Yaskawa INFORM job: DEMO_ROOF_SIDE_0625_3PAINT_33.JBI

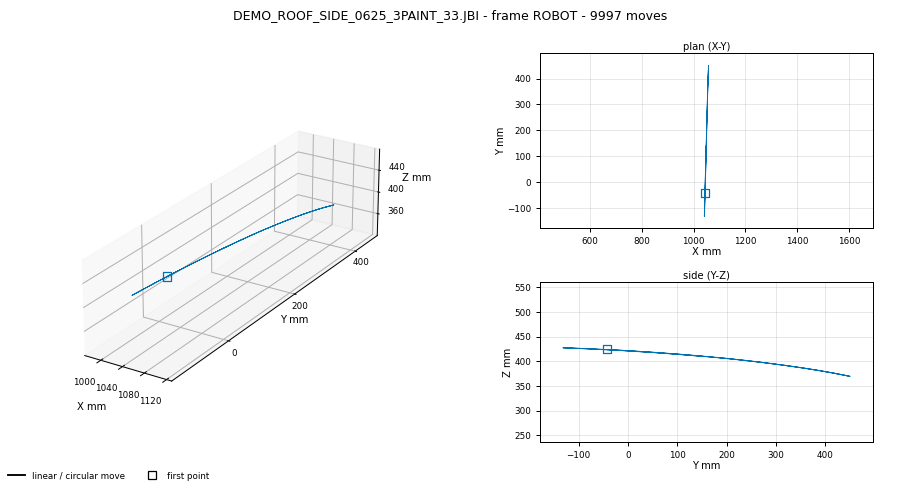
[picture p0: tool path of DEMO_ROOF_SIDE_0625_3PAINT_33.JBI in frame ROBOT, 9997 of 9997 moves have a stored position in this frame; points joined in program order, loops and branches not executed]
/JOB
//NAME DEMO_ROOF_SIDE_0625_3PAINT33
//POS
///NPOS 9997,0,0,0,0,0
///TOOL 0
///USER 0
///POSTYPE ROBOT
///RECTAN
///RCONF 1,0,0,0,0,0,0,0,0,0,0,0,0,0,0,0,0,0,0,0,0,0,0,0
C00000=1044.636,-42.308,424.466,169.630,34.372,156.485
C00001=1044.642,-42.058,424.454,169.632,34.373,156.485
C00002=1044.648,-41.809,424.441,169.634,34.375,156.485
C00003=1044.655,-41.560,424.428,169.636,34.375,156.486
C00004=1044.661,-41.310,424.415,169.638,34.376,156.486
C00005=1044.667,-41.061,424.402,169.640,34.377,156.486
C00006=1044.674,-40.810,424.389,169.642,34.378,156.486
C00007=1044.680,-40.561,424.376,169.645,34.379,156.486
C00008=1044.687,-40.311,424.364,169.647,34.380,156.486
C00009=1044.693,-40.062,424.351,169.649,34.381,156.486
C00010=1044.699,-39.813,424.337,169.651,34.382,156.486
C00011=1044.706,-39.562,424.324,169.653,34.383,156.486
C00012=1044.712,-39.313,424.311,169.656,34.384,156.487
C00013=1044.718,-39.063,424.299,169.658,34.385,156.487
C00014=1044.725,-38.814,424.286,169.660,34.385,156.487
C00015=1044.731,-38.565,424.273,169.662,34.387,156.487
C00016=1044.738,-38.314,424.260,169.664,34.388,156.487
C00017=1044.744,-38.065,424.246,169.666,34.389,156.487
C00018=1044.749,-37.816,424.233,169.668,34.390,156.487
C00019=1044.755,-37.566,424.219,169.670,34.391,156.488
C00020=1044.761,-37.316,424.207,169.672,34.392,156.488
C00021=1044.768,-37.067,424.193,169.674,34.393,156.488
C00022=1044.774,-36.817,424.180,169.677,34.394,156.488
C00023=1044.781,-36.568,424.167,169.679,34.395,156.488
C00024=1044.787,-36.318,424.154,169.681,34.396,156.488
C00025=1044.793,-36.069,424.141,169.683,34.398,156.488
C00026=1044.800,-35.819,424.127,169.685,34.398,156.489
C00027=1044.806,-35.538,424.113,169.687,34.400,156.489
C00028=1044.813,-35.257,424.097,169.689,34.401,156.489
C00029=1044.820,-34.977,424.083,169.692,34.402,156.489
C00030=1044.828,-34.695,424.068,169.694,34.403,156.489
C00031=1044.834,-34.446,424.055,169.696,34.405,156.489
C00032=1044.840,-34.197,424.042,169.698,34.405,156.489
C00033=1044.846,-33.947,424.028,169.700,34.407,156.490
C00034=1044.852,-33.697,424.014,169.702,34.407,156.490
C00035=1044.858,-33.448,424.002,169.704,34.409,156.490
C00036=1044.864,-33.198,423.988,169.706,34.410,156.490
C00037=1044.871,-32.949,423.975,169.708,34.411,156.490
C00038=1044.878,-32.699,423.961,169.710,34.412,156.490
C00039=1044.884,-32.450,423.948,169.712,34.413,156.491
C00040=1044.890,-32.200,423.935,169.714,34.414,156.491
C00041=1044.897,-31.951,423.921,169.716,34.415,156.491
C00042=1044.903,-31.701,423.908,169.718,34.416,156.491
C00043=1044.909,-31.452,423.895,169.720,34.417,156.491
C00044=1044.915,-31.201,423.881,169.722,34.418,156.491
C00045=1044.921,-30.952,423.868,169.724,34.419,156.491
C00046=1044.927,-30.703,423.855,169.726,34.420,156.491
C00047=1044.934,-30.453,423.841,169.728,34.422,156.492
C00048=1044.940,-30.203,423.828,169.730,34.422,156.492
C00049=1044.947,-29.954,423.814,169.732,34.424,156.492
C00050=1044.953,-29.704,423.801,169.734,34.424,156.492
C00051=1044.960,-29.455,423.788,169.736,34.426,156.492
C00052=1044.966,-29.206,423.774,169.739,34.427,156.492
C00053=1044.972,-28.955,423.760,169.741,34.428,156.493
C00054=1044.978,-28.706,423.747,169.743,34.429,156.493
C00055=1044.984,-28.457,423.733,169.745,34.430,156.493
C00056=1044.991,-28.207,423.720,169.748,34.431,156.493
C00057=1044.997,-27.958,423.707,169.750,34.432,156.493
C00058=1045.004,-27.708,423.693,169.752,34.434,156.493
C00059=1045.010,-27.458,423.680,169.754,34.434,156.493
C00060=1045.017,-27.209,423.666,169.756,34.436,156.494
C00061=1045.023,-26.959,423.652,169.758,34.436,156.494
C00062=1045.029,-26.710,423.639,169.760,34.438,156.494
C00063=1045.035,-26.461,423.625,169.762,34.439,156.494
C00064=1045.042,-26.211,423.611,169.763,34.440,156.494
C00065=1045.048,-25.961,423.597,169.765,34.441,156.494
C00066=1045.054,-25.712,423.584,169.767,34.443,156.495
C00067=1045.060,-25.462,423.570,169.769,34.444,156.495
C00068=1045.066,-25.213,423.557,169.771,34.445,156.495
C00069=1045.073,-24.963,423.543,169.773,34.446,156.495
C00070=1045.079,-24.714,423.528,169.775,34.447,156.495
C00071=1045.085,-24.464,423.515,169.777,34.448,156.495
C00072=1045.091,-24.214,423.501,169.779,34.450,156.496
C00073=1045.097,-23.965,423.488,169.781,34.451,156.496
C00074=1045.104,-23.715,423.474,169.783,34.452,156.496
C00075=1045.110,-23.465,423.460,169.785,34.453,156.496
C00076=1045.116,-23.217,423.446,169.787,34.454,156.496
C00077=1045.123,-22.967,423.433,169.789,34.456,156.496
C00078=1045.128,-22.717,423.419,169.791,34.457,156.497
C00079=1045.135,-22.467,423.405,169.793,34.458,156.497
C00080=1045.141,-22.218,423.390,169.795,34.459,156.497
C00081=1045.148,-21.968,423.377,169.797,34.461,156.497
C00082=1045.154,-21.719,423.364,169.799,34.461,156.497
C00083=1045.160,-21.469,423.350,169.801,34.463,156.497
C00084=1045.167,-21.220,423.335,169.804,34.464,156.498
C00085=1045.172,-20.970,423.321,169.806,34.465,156.498
C00086=1045.179,-20.720,423.308,169.808,34.466,156.498
C00087=1045.186,-20.472,423.294,169.810,34.468,156.498
C00088=1045.192,-20.222,423.280,169.812,34.469,156.498
C00089=1045.198,-19.972,423.266,169.814,34.470,156.498
C00090=1045.204,-19.723,423.251,169.816,34.471,156.499
C00091=1045.211,-19.441,423.236,169.818,34.472,156.499
C00092=1045.218,-19.159,423.220,169.820,34.474,156.499
C00093=1045.225,-18.878,423.205,169.822,34.475,156.499
C00094=1045.232,-18.596,423.189,169.824,34.477,156.499
C00095=1045.239,-18.347,423.175,169.826,34.478,156.500
C00096=1045.245,-18.097,423.161,169.828,34.479,156.500
C00097=1045.252,-17.848,423.147,169.830,34.480,156.500
C00098=1045.258,-17.598,423.133,169.832,34.481,156.500
C00099=1045.264,-17.348,423.119,169.834,34.482,156.500
C00100=1045.271,-17.099,423.105,169.836,34.484,156.500
C00101=1045.277,-16.849,423.091,169.838,34.485,156.501
C00102=1045.284,-16.600,423.077,169.840,34.486,156.501
C00103=1045.290,-16.350,423.063,169.842,34.487,156.501
C00104=1045.296,-16.101,423.049,169.844,34.488,156.501
C00105=1045.303,-15.851,423.035,169.846,34.490,156.501
C00106=1045.308,-15.602,423.021,169.848,34.491,156.502
C00107=1045.316,-15.352,423.007,169.850,34.492,156.502
C00108=1045.322,-15.102,422.993,169.852,34.493,156.502
C00109=1045.327,-14.853,422.978,169.854,34.495,156.502
C00110=1045.334,-14.603,422.964,169.855,34.496,156.502
C00111=1045.340,-14.354,422.950,169.858,34.497,156.502
C00112=1045.346,-14.104,422.936,169.860,34.499,156.503
C00113=1045.353,-13.855,422.922,169.862,34.500,156.503
C00114=1045.359,-13.605,422.907,169.864,34.501,156.503
C00115=1045.365,-13.356,422.893,169.866,34.502,156.503
C00116=1045.372,-13.107,422.878,169.868,34.503,156.503
C00117=1045.378,-12.856,422.864,169.870,34.505,156.504
C00118=1045.383,-12.607,422.850,169.872,34.506,156.504
C00119=1045.390,-12.357,422.836,169.874,34.508,156.504
C00120=1045.396,-12.109,422.821,169.876,34.509,156.504
C00121=1045.402,-11.859,422.806,169.877,34.510,156.504
C00122=1045.409,-11.610,422.793,169.879,34.512,156.505
C00123=1045.415,-11.360,422.778,169.881,34.512,156.505
C00124=1045.421,-11.110,422.764,169.883,34.514,156.505
C00125=1045.428,-10.861,422.750,169.885,34.515,156.505
C00126=1045.434,-10.611,422.735,169.887,34.516,156.505
C00127=1045.440,-10.361,422.721,169.889,34.518,156.505
C00128=1045.447,-10.112,422.707,169.891,34.519,156.506
C00129=1045.453,-9.863,422.692,169.893,34.521,156.506
C00130=1045.459,-9.613,422.678,169.895,34.522,156.506
C00131=1045.466,-9.364,422.664,169.896,34.523,156.506
C00132=1045.472,-9.114,422.649,169.898,34.525,156.507
C00133=1045.478,-8.865,422.634,169.900,34.525,156.507
C00134=1045.484,-8.615,422.620,169.903,34.527,156.507
C00135=1045.491,-8.366,422.606,169.905,34.528,156.507
C00136=1045.497,-8.117,422.591,169.907,34.529,156.507
C00137=1045.503,-7.866,422.577,169.909,34.531,156.507
C00138=1045.510,-7.617,422.562,169.911,34.532,156.508
C00139=1045.516,-7.368,422.548,169.913,34.534,156.508
C00140=1045.522,-7.118,422.533,169.914,34.535,156.508
C00141=1045.528,-6.868,422.519,169.916,34.536,156.508
C00142=1045.535,-6.620,422.505,169.918,34.537,156.508
C00143=1045.541,-6.370,422.490,169.920,34.538,156.509
C00144=1045.548,-6.120,422.475,169.922,34.540,156.509
C00145=1045.555,-5.871,422.460,169.924,34.541,156.509
C00146=1045.560,-5.621,422.447,169.926,34.542,156.509
C00147=1045.566,-5.372,422.432,169.928,34.544,156.509
C00148=1045.573,-5.122,422.417,169.929,34.545,156.510
C00149=1045.580,-4.873,422.402,169.931,34.546,156.510
C00150=1045.586,-4.624,422.388,169.933,34.548,156.510
C00151=1045.592,-4.373,422.373,169.935,34.549,156.510
C00152=1045.598,-4.124,422.359,169.937,34.551,156.510
C00153=1045.605,-3.875,422.345,169.939,34.551,156.510
C00154=1045.611,-3.625,422.330,169.941,34.553,156.511
C00155=1045.618,-3.342,422.313,169.943,34.555,156.511
C00156=1045.626,-3.059,422.296,169.946,34.556,156.511
C00157=1045.632,-2.775,422.279,169.948,34.557,156.511
C00158=1045.639,-2.492,422.262,169.950,34.559,156.512
C00159=1045.646,-2.243,422.247,169.952,34.561,156.512
C00160=1045.651,-1.994,422.233,169.954,34.562,156.512
C00161=1045.658,-1.744,422.218,169.956,34.563,156.512
C00162=1045.664,-1.495,422.203,169.957,34.565,156.513
C00163=1045.671,-1.245,422.188,169.959,34.566,156.513
C00164=1045.676,-0.996,422.173,169.961,34.567,156.513
C00165=1045.683,-0.746,422.158,169.963,34.569,156.513
C00166=1045.689,-0.497,422.143,169.965,34.570,156.513
C00167=1045.696,-0.247,422.128,169.967,34.572,156.514
C00168=1045.701,0.002,422.114,169.968,34.573,156.514
C00169=1045.708,0.252,422.099,169.970,34.575,156.514
C00170=1045.713,0.502,422.083,169.972,34.576,156.514
C00171=1045.720,0.751,422.068,169.974,34.578,156.515
C00172=1045.726,1.000,422.054,169.976,34.579,156.515
C00173=1045.732,1.250,422.039,169.978,34.580,156.515
C00174=1045.738,1.500,422.024,169.979,34.582,156.515
C00175=1045.745,1.749,422.009,169.982,34.583,156.515
C00176=1045.750,1.998,421.994,169.984,34.584,156.516
C00177=1045.757,2.248,421.979,169.986,34.586,156.516
C00178=1045.763,2.497,421.965,169.988,34.588,156.516
C00179=1045.770,2.746,421.949,169.989,34.589,156.516
C00180=1045.776,2.996,421.934,169.991,34.590,156.517
C00181=1045.783,3.246,421.919,169.993,34.592,156.517
C00182=1045.788,3.495,421.904,169.995,34.593,156.517
C00183=1045.795,3.744,421.889,169.997,34.594,156.517
C00184=1045.801,3.994,421.874,169.999,34.596,156.517
C00185=1045.807,4.244,421.859,170.000,34.597,156.518
C00186=1045.814,4.493,421.843,170.002,34.598,156.518
C00187=1045.820,4.743,421.828,170.004,34.600,156.518
C00188=1045.826,4.992,421.814,170.006,34.601,156.518
C00189=1045.832,5.241,421.799,170.008,34.603,156.518
C00190=1045.839,5.491,421.784,170.009,34.604,156.519
C00191=1045.845,5.740,421.768,170.011,34.606,156.519
C00192=1045.852,5.990,421.753,170.013,34.607,156.519
C00193=1045.858,6.239,421.738,170.016,34.608,156.519
C00194=1045.864,6.489,421.723,170.018,34.610,156.520
C00195=1045.869,6.738,421.708,170.020,34.611,156.520
C00196=1045.876,6.987,421.693,170.021,34.612,156.520
C00197=1045.882,7.237,421.678,170.023,34.614,156.520
C00198=1045.889,7.487,421.663,170.025,34.615,156.520
C00199=1045.895,7.736,421.648,170.027,34.617,156.521
C00200=1045.902,7.985,421.632,170.029,34.618,156.521
C00201=1045.908,8.235,421.617,170.030,34.620,156.521
C00202=1045.915,8.485,421.602,170.032,34.621,156.521
C00203=1045.921,8.734,421.586,170.034,34.623,156.522
C00204=1045.927,8.984,421.571,170.036,34.624,156.522
C00205=1045.933,9.233,421.556,170.038,34.625,156.522
C00206=1045.940,9.482,421.540,170.039,34.627,156.522
C00207=1045.946,9.731,421.526,170.041,34.628,156.522
C00208=1045.952,9.981,421.511,170.043,34.629,156.523
C00209=1045.959,10.230,421.495,170.045,34.631,156.523
C00210=1045.965,10.480,421.480,170.047,34.633,156.523
C00211=1045.971,10.730,421.465,170.049,34.634,156.523
C00212=1045.978,10.979,421.449,170.051,34.635,156.524
C00213=1045.984,11.228,421.434,170.053,34.637,156.524
C00214=1045.990,11.478,421.419,170.055,34.638,156.524
C00215=1045.997,11.727,421.403,170.057,34.639,156.524
C00216=1046.004,11.977,421.388,170.058,34.641,156.524
C00217=1046.010,12.226,421.373,170.060,34.642,156.525
C00218=1046.016,12.476,421.357,170.062,34.643,156.525
C00219=1046.023,12.761,421.340,170.064,34.645,156.525
C00220=1046.031,13.046,421.322,170.066,34.647,156.525
C00221=1046.038,13.331,421.305,170.068,34.648,156.526
C00222=1046.045,13.616,421.287,170.070,34.650,156.526
C00223=1046.052,13.865,421.272,170.072,34.651,156.526
C00224=1046.058,14.115,421.257,170.074,34.653,156.526
C00225=1046.065,14.364,421.241,170.076,34.654,156.526
C00226=1046.070,14.614,421.226,170.077,34.655,156.527
C00227=1046.077,14.863,421.210,170.080,34.657,156.527
C00228=1046.083,15.113,421.194,170.082,34.659,156.527
C00229=1046.090,15.362,421.179,170.084,34.660,156.527
C00230=1046.096,15.611,421.163,170.085,34.661,156.528
C00231=1046.102,15.861,421.148,170.087,34.663,156.528
C00232=1046.109,16.110,421.132,170.089,34.665,156.528
C00233=1046.114,16.360,421.117,170.091,34.666,156.528
C00234=1046.121,16.609,421.101,170.092,34.667,156.529
C00235=1046.127,16.859,421.086,170.094,34.669,156.529
C00236=1046.133,17.108,421.070,170.096,34.671,156.529
C00237=1046.140,17.357,421.054,170.098,34.672,156.529
C00238=1046.146,17.607,421.038,170.099,34.673,156.530
C00239=1046.152,17.856,421.023,170.101,34.675,156.530
C00240=1046.159,18.107,421.008,170.103,34.677,156.530
C00241=1046.165,18.356,420.991,170.105,34.678,156.530
C00242=1046.172,18.605,420.976,170.106,34.679,156.530
C00243=1046.177,18.855,420.960,170.109,34.681,156.531
C00244=1046.184,19.104,420.944,170.111,34.682,156.531
C00245=1046.191,19.353,420.929,170.113,34.684,156.531
C00246=1046.197,19.603,420.913,170.114,34.685,156.531
C00247=1046.203,19.852,420.898,170.116,34.687,156.532
C00248=1046.209,20.101,420.881,170.118,34.688,156.532
C00249=1046.216,20.351,420.866,170.120,34.690,156.532
C00250=1046.221,20.600,420.850,170.121,34.691,156.532
C00251=1046.228,20.849,420.834,170.123,34.693,156.533
C00252=1046.234,21.099,420.818,170.125,34.695,156.533
C00253=1046.240,21.349,420.803,170.127,34.696,156.533
C00254=1046.246,21.598,420.787,170.128,34.697,156.533
C00255=1046.253,21.848,420.770,170.130,34.699,156.534
C00256=1046.260,22.097,420.755,170.132,34.700,156.534
C00257=1046.265,22.347,420.739,170.134,34.702,156.534
C00258=1046.272,22.596,420.723,170.135,34.703,156.534
C00259=1046.278,22.845,420.707,170.138,34.705,156.535
C00260=1046.285,23.094,420.692,170.140,34.706,156.535
C00261=1046.291,23.344,420.675,170.142,34.708,156.535
C00262=1046.296,23.594,420.660,170.143,34.709,156.535
C00263=1046.303,23.843,420.644,170.145,34.711,156.536
C00264=1046.310,24.093,420.627,170.147,34.712,156.536
C00265=1046.316,24.342,420.612,170.148,34.714,156.536
C00266=1046.322,24.591,420.596,170.150,34.716,156.536
C00267=1046.329,24.841,420.581,170.152,34.717,156.537
C00268=1046.334,25.090,420.564,170.154,34.718,156.537
C00269=1046.340,25.339,420.548,170.155,34.720,156.537
C00270=1046.347,25.588,420.532,170.157,34.722,156.537
C00271=1046.354,25.839,420.516,170.159,34.723,156.538
C00272=1046.360,26.088,420.500,170.161,34.724,156.538
C00273=1046.366,26.337,420.484,170.163,34.726,156.538
C00274=1046.373,26.586,420.468,170.165,34.728,156.538
C00275=1046.379,26.835,420.452,170.167,34.729,156.538
C00276=1046.385,27.085,420.436,170.168,34.730,156.539
C00277=1046.392,27.335,420.420,170.170,34.732,156.539
C00278=1046.398,27.584,420.404,170.172,34.734,156.539
C00279=1046.404,27.834,420.388,170.174,34.735,156.539
C00280=1046.410,28.083,420.372,170.175,34.737,156.540
C00281=1046.416,28.332,420.356,170.177,34.738,156.540
C00282=1046.423,28.582,420.339,170.179,34.740,156.540
C00283=1046.430,28.868,420.321,170.181,34.741,156.541
C00284=1046.438,29.155,420.302,170.183,34.743,156.541
C00285=1046.445,29.440,420.284,170.185,34.745,156.541
C00286=1046.451,29.727,420.265,170.187,34.747,156.541
C00287=1046.458,29.977,420.249,170.189,34.749,156.542
C00288=1046.464,30.226,420.233,170.191,34.750,156.542
C00289=1046.470,30.476,420.217,170.193,34.751,156.542
C00290=1046.476,30.725,420.200,170.194,34.753,156.542
C00291=1046.482,30.974,420.183,170.196,34.755,156.543
C00292=1046.490,31.224,420.167,170.198,34.756,156.543
C00293=1046.496,31.473,420.151,170.200,34.758,156.543
C00294=1046.502,31.722,420.135,170.201,34.759,156.543
C00295=1046.507,31.972,420.119,170.203,34.761,156.544
C00296=1046.514,32.222,420.102,170.205,34.763,156.544
C00297=1046.521,32.471,420.086,170.206,34.764,156.544
C00298=1046.527,32.720,420.070,170.208,34.766,156.545
C00299=1046.533,32.969,420.054,170.210,34.767,156.545
C00300=1046.539,33.219,420.037,170.212,34.768,156.545
C00301=1046.545,33.468,420.020,170.214,34.770,156.545
C00302=1046.552,33.717,420.005,170.216,34.772,156.545
C00303=1046.558,33.967,419.988,170.218,34.774,156.546
C00304=1046.565,34.217,419.972,170.219,34.775,156.546
C00305=1046.571,34.466,419.956,170.221,34.776,156.546
C00306=1046.577,34.715,419.939,170.223,34.778,156.547
C00307=1046.583,34.964,419.922,170.224,34.780,156.547
C00308=1046.590,35.214,419.906,170.226,34.781,156.547
C00309=1046.596,35.463,419.890,170.228,34.783,156.547
C00310=1046.602,35.713,419.874,170.229,34.784,156.548
C00311=1046.609,35.963,419.857,170.231,34.786,156.548
C00312=1046.615,36.211,419.840,170.233,34.788,156.548
C00313=1046.621,36.461,419.824,170.236,34.789,156.548
C00314=1046.628,36.710,419.808,170.237,34.791,156.549
C00315=1046.634,36.960,419.792,170.239,34.792,156.549
C00316=1046.640,37.208,419.775,170.241,34.793,156.549
C00317=1046.646,37.458,419.758,170.242,34.795,156.549
C00318=1046.653,37.708,419.742,170.244,34.797,156.550
C00319=1046.659,37.957,419.725,170.246,34.799,156.550
C00320=1046.665,38.206,419.709,170.247,34.800,156.550
C00321=1046.671,38.456,419.692,170.249,34.801,156.550
C00322=1046.677,38.705,419.676,170.251,34.803,156.551
C00323=1046.684,38.954,419.659,170.252,34.805,156.551
C00324=1046.690,39.204,419.642,170.254,34.807,156.551
C00325=1046.697,39.453,419.625,170.256,34.808,156.551
C00326=1046.702,39.702,419.609,170.258,34.810,156.552
C00327=1046.709,39.952,419.592,170.260,34.811,156.552
C00328=1046.715,40.201,419.575,170.262,34.813,156.552
C00329=1046.720,40.451,419.558,170.263,34.814,156.553
C00330=1046.727,40.701,419.542,170.265,34.816,156.553
C00331=1046.733,40.949,419.525,170.267,34.818,156.553
C00332=1046.739,41.199,419.509,170.268,34.820,156.553
C00333=1046.746,41.448,419.491,170.270,34.821,156.554
C00334=1046.752,41.698,419.475,170.272,34.822,156.554
C00335=1046.758,41.947,419.459,170.273,34.824,156.554
C00336=1046.765,42.196,419.441,170.275,34.825,156.554
C00337=1046.771,42.446,419.425,170.277,34.827,156.555
C00338=1046.777,42.694,419.408,170.279,34.829,156.555
C00339=1046.784,42.944,419.391,170.281,34.831,156.555
C00340=1046.790,43.193,419.375,170.283,34.832,156.555
C00341=1046.796,43.443,419.358,170.285,34.834,156.556
C00342=1046.802,43.692,419.340,170.286,34.835,156.556
C00343=1046.808,43.942,419.324,170.288,34.837,156.556
C00344=1046.815,44.191,419.307,170.289,34.839,156.557
C00345=1046.820,44.441,419.290,170.291,34.840,156.557
C00346=1046.826,44.689,419.273,170.293,34.842,156.557
C00347=1046.833,44.977,419.253,170.295,34.844,156.558
C00348=1046.840,45.263,419.233,170.297,34.846,156.558
C00349=1046.848,45.549,419.215,170.298,34.848,156.558
C00350=1046.855,45.835,419.195,170.301,34.850,156.558
C00351=1046.861,46.085,419.178,170.303,34.852,156.559
C00352=1046.867,46.334,419.161,170.305,34.854,156.559
C00353=1046.873,46.583,419.144,170.306,34.855,156.559
C00354=1046.879,46.833,419.126,170.308,34.857,156.560
C00355=1046.885,47.082,419.109,170.310,34.858,156.560
C00356=1046.891,47.331,419.093,170.311,34.860,156.560
C00357=1046.897,47.581,419.075,170.313,34.861,156.560
C00358=1046.904,47.830,419.058,170.314,34.863,156.561
C00359=1046.910,48.080,419.042,170.316,34.865,156.561
C00360=1046.916,48.329,419.024,170.318,34.867,156.561
C00361=1046.922,48.578,419.007,170.320,34.868,156.562
C00362=1046.928,48.827,418.990,170.322,34.870,156.562
C00363=1046.934,49.076,418.973,170.324,34.872,156.562
C00364=1046.941,49.326,418.956,170.325,34.873,156.562
C00365=1046.947,49.575,418.939,170.327,34.875,156.563
C00366=1046.953,49.825,418.921,170.329,34.876,156.563
C00367=1046.959,50.074,418.904,170.330,34.878,156.563
C00368=1046.966,50.324,418.888,170.332,34.880,156.564
C00369=1046.971,50.573,418.870,170.334,34.882,156.564
C00370=1046.978,50.822,418.853,170.335,34.883,156.564
C00371=1046.984,51.071,418.836,170.337,34.885,156.564
C00372=1046.990,51.321,418.819,170.340,34.887,156.565
C00373=1046.996,51.570,418.802,170.341,34.888,156.565
C00374=1047.003,51.819,418.784,170.343,34.890,156.565
C00375=1047.009,52.068,418.767,170.344,34.891,156.565
C00376=1047.015,52.318,418.751,170.346,34.893,156.566
C00377=1047.021,52.568,418.733,170.348,34.895,156.566
C00378=1047.028,52.817,418.715,170.349,34.896,156.566
C00379=1047.034,53.066,418.698,170.351,34.898,156.567
C00380=1047.040,53.315,418.680,170.353,34.900,156.567
C00381=1047.046,53.565,418.664,170.354,34.902,156.567
C00382=1047.053,53.814,418.647,170.356,34.903,156.567
C00383=1047.058,54.063,418.629,170.359,34.905,156.568
C00384=1047.065,54.313,418.612,170.360,34.906,156.568
C00385=1047.071,54.562,418.594,170.362,34.908,156.568
C00386=1047.078,54.811,418.577,170.364,34.909,156.568
C00387=1047.084,55.060,418.560,170.365,34.911,156.569
C00388=1047.090,55.310,418.543,170.367,34.913,156.569
C00389=1047.096,55.559,418.526,170.369,34.915,156.569
C00390=1047.103,55.808,418.508,170.370,34.916,156.570
C00391=1047.109,56.058,418.491,170.372,34.918,156.570
C00392=1047.115,56.307,418.474,170.374,34.919,156.570
C00393=1047.121,56.557,418.456,170.375,34.921,156.570
C00394=1047.128,56.805,418.439,170.377,34.922,156.571
C00395=1047.134,57.055,418.421,170.379,34.924,156.571
C00396=1047.140,57.304,418.404,170.381,34.926,156.571
C00397=1047.147,57.553,418.386,170.383,34.928,156.572
C00398=1047.153,57.804,418.369,170.384,34.929,156.572
C00399=1047.159,58.052,418.352,170.386,34.931,156.572
C00400=1047.166,58.302,418.335,170.388,34.932,156.572
C00401=1047.171,58.551,418.317,170.389,34.934,156.573
C00402=1047.178,58.800,418.300,170.391,34.935,156.573
C00403=1047.184,59.050,418.282,170.393,34.937,156.573
C00404=1047.190,59.299,418.265,170.394,34.939,156.573
C00405=1047.197,59.548,418.247,170.397,34.941,156.574
C00406=1047.203,59.798,418.230,170.399,34.942,156.574
C00407=1047.210,60.047,418.213,170.400,34.944,156.574
C00408=1047.216,60.296,418.195,170.402,34.945,156.575
C00409=1047.223,60.546,418.178,170.404,34.947,156.575
C00410=1047.228,60.795,418.160,170.405,34.948,156.575
C00411=1047.236,61.081,418.140,170.407,34.950,156.575
C00412=1047.244,61.366,418.120,170.409,34.952,156.576
C00413=1047.251,61.652,418.100,170.411,34.954,156.576
C00414=1047.258,61.939,418.079,170.413,34.956,156.576
C00415=1047.264,62.188,418.062,170.415,34.958,156.577
C00416=1047.271,62.438,418.044,170.417,34.959,156.577
C00417=1047.278,62.687,418.027,170.419,34.961,156.577
C00418=1047.283,62.936,418.010,170.420,34.963,156.578
C00419=1047.290,63.185,417.992,170.422,34.964,156.578
C00420=1047.296,63.435,417.974,170.424,34.966,156.578
C00421=1047.303,63.684,417.956,170.425,34.967,156.578
C00422=1047.309,63.933,417.939,170.427,34.969,156.579
C00423=1047.316,64.182,417.921,170.429,34.970,156.579
C00424=1047.322,64.432,417.903,170.430,34.972,156.579
C00425=1047.327,64.681,417.886,170.432,34.974,156.579
C00426=1047.334,64.931,417.868,170.434,34.976,156.580
C00427=1047.341,65.180,417.850,170.436,34.978,156.580
C00428=1047.346,65.429,417.832,170.438,34.979,156.580
C00429=1047.352,65.679,417.814,170.440,34.981,156.581
C00430=1047.359,65.928,417.797,170.441,34.982,156.581
C00431=1047.365,66.177,417.779,170.443,34.984,156.581
C00432=1047.371,66.426,417.761,170.444,34.986,156.581
C00433=1047.378,66.676,417.743,170.446,34.987,156.582
C00434=1047.384,66.925,417.725,170.448,34.989,156.582
C00435=1047.389,67.174,417.708,170.449,34.990,156.582
C00436=1047.396,67.423,417.689,170.451,34.992,156.583
C00437=1047.403,67.673,417.672,170.454,34.994,156.583
C00438=1047.408,67.922,417.654,170.455,34.996,156.583
C00439=1047.415,68.171,417.636,170.457,34.998,156.583
C00440=1047.421,68.421,417.618,170.458,34.999,156.584
C00441=1047.428,68.670,417.600,170.460,35.001,156.584
C00442=1047.433,68.919,417.582,170.462,35.003,156.584
C00443=1047.440,69.168,417.564,170.463,35.004,156.585
C00444=1047.446,69.418,417.546,170.465,35.006,156.585
C00445=1047.453,69.667,417.528,170.467,35.008,156.585
C00446=1047.458,69.916,417.511,170.468,35.009,156.585
C00447=1047.465,70.166,417.493,170.471,35.011,156.586
C00448=1047.471,70.415,417.474,170.473,35.013,156.586
C00449=1047.476,70.664,417.457,170.474,35.014,156.586
C00450=1047.483,70.913,417.438,170.476,35.016,156.587
C00451=1047.489,71.163,417.420,170.477,35.018,156.587
C00452=1047.495,71.413,417.402,170.479,35.019,156.587
C00453=1047.502,71.661,417.384,170.481,35.021,156.588
C00454=1047.508,71.910,417.366,170.482,35.023,156.588
C00455=1047.514,72.159,417.348,170.484,35.025,156.588
C00456=1047.520,72.409,417.330,170.486,35.027,156.588
C00457=1047.526,72.658,417.312,170.488,35.028,156.589
C00458=1047.532,72.907,417.294,170.490,35.030,156.589
C00459=1047.539,73.157,417.275,170.491,35.032,156.589
C00460=1047.545,73.406,417.257,170.493,35.034,156.590
C00461=1047.551,73.655,417.238,170.495,35.035,156.590
C00462=1047.557,73.904,417.221,170.496,35.037,156.590
C00463=1047.563,74.154,417.202,170.498,35.039,156.591
C00464=1047.569,74.403,417.184,170.500,35.040,156.591
C00465=1047.576,74.652,417.166,170.501,35.042,156.591
C00466=1047.583,74.902,417.148,170.504,35.044,156.591
C00467=1047.588,75.150,417.130,170.505,35.045,156.592
C00468=1047.595,75.400,417.112,170.507,35.047,156.592
C00469=1047.601,75.649,417.093,170.509,35.049,156.592
C00470=1047.607,75.899,417.075,170.510,35.050,156.593
C00471=1047.614,76.148,417.057,170.512,35.052,156.593
C00472=1047.620,76.398,417.039,170.514,35.054,156.593
C00473=1047.626,76.646,417.021,170.515,35.056,156.594
C00474=1047.632,76.895,417.002,170.517,35.057,156.594
C00475=1047.639,77.182,416.982,170.519,35.059,156.594
C00476=1047.646,77.468,416.960,170.522,35.061,156.595
C00477=1047.653,77.753,416.939,170.523,35.063,156.595
C00478=1047.660,78.039,416.918,170.525,35.065,156.595
C00479=1047.667,78.288,416.899,170.527,35.067,156.596
C00480=1047.673,78.538,416.881,170.529,35.068,156.596
C00481=1047.679,78.786,416.863,170.530,35.070,156.596
C00482=1047.684,79.036,416.844,170.532,35.072,156.596
C00483=1047.691,79.286,416.826,170.533,35.074,156.597
C00484=1047.697,79.535,416.807,170.535,35.075,156.597
C00485=1047.703,79.784,416.789,170.538,35.077,156.597
C00486=1047.710,80.033,416.770,170.539,35.079,156.598
C00487=1047.715,80.282,416.752,170.541,35.081,156.598
C00488=1047.721,80.531,416.733,170.543,35.083,156.598
C00489=1047.728,80.781,416.715,170.544,35.084,156.599
C00490=1047.734,81.030,416.696,170.546,35.086,156.599
C00491=1047.740,81.279,416.678,170.547,35.088,156.599
C00492=1047.746,81.529,416.659,170.549,35.090,156.599
C00493=1047.752,81.778,416.640,170.551,35.092,156.600
C00494=1047.759,82.027,416.621,170.553,35.093,156.600
C00495=1047.764,82.276,416.604,170.555,35.095,156.600
C00496=1047.771,82.525,416.585,170.556,35.097,156.601
C00497=1047.777,82.774,416.567,170.558,35.099,156.601
C00498=1047.783,83.024,416.547,170.560,35.100,156.601
C00499=1047.789,83.273,416.529,170.561,35.102,156.602
C00500=1047.796,83.522,416.510,170.563,35.104,156.602
C00501=1047.802,83.772,416.492,170.565,35.106,156.602
C00502=1047.807,84.021,416.473,170.566,35.107,156.603
C00503=1047.814,84.270,416.454,170.569,35.109,156.603
C00504=1047.820,84.519,416.436,170.571,35.111,156.603
C00505=1047.826,84.768,416.417,170.572,35.113,156.603
C00506=1047.832,85.017,416.399,170.574,35.115,156.604
C00507=1047.838,85.266,416.379,170.575,35.116,156.604
C00508=1047.845,85.516,416.361,170.577,35.118,156.604
C00509=1047.851,85.765,416.343,170.579,35.120,156.605
C00510=1047.857,86.014,416.324,170.580,35.122,156.605
C00511=1047.863,86.264,416.305,170.582,35.123,156.605
C00512=1047.869,86.513,416.286,170.585,35.125,156.606
C00513=1047.876,86.762,416.268,170.586,35.127,156.606
C00514=1047.882,87.011,416.249,170.588,35.128,156.606
C00515=1047.888,87.261,416.230,170.589,35.130,156.607
C00516=1047.894,87.510,416.211,170.591,35.132,156.607
C00517=1047.901,87.759,416.192,170.593,35.133,156.607
C00518=1047.907,88.008,416.174,170.594,35.135,156.607
C00519=1047.913,88.257,416.155,170.596,35.137,156.608
C00520=1047.919,88.507,416.136,170.598,35.139,156.608
C00521=1047.926,88.756,416.117,170.600,35.140,156.608
C00522=1047.932,89.005,416.099,170.602,35.142,156.609
C00523=1047.938,89.254,416.079,170.604,35.144,156.609
C00524=1047.944,89.503,416.061,170.605,35.145,156.609
C00525=1047.951,89.753,416.042,170.607,35.147,156.610
C00526=1047.957,90.002,416.023,170.609,35.149,156.610
C00527=1047.963,90.251,416.004,170.610,35.150,156.610
C00528=1047.969,90.500,415.986,170.612,35.152,156.610
C00529=1047.975,90.750,415.966,170.613,35.154,156.611
C00530=1047.981,90.999,415.948,170.616,35.156,156.611
C00531=1047.987,91.248,415.928,170.618,35.158,156.611
C00532=1047.993,91.497,415.910,170.619,35.159,156.612
C00533=1047.999,91.747,415.891,170.621,35.161,156.612
C00534=1048.006,91.995,415.871,170.623,35.163,156.612
C00535=1048.011,92.245,415.852,170.624,35.165,156.613
C00536=1048.018,92.494,415.833,170.626,35.167,156.613
C00537=1048.024,92.743,415.814,170.627,35.168,156.613
C00538=1048.030,92.992,415.795,170.630,35.170,156.614
C00539=1048.037,93.278,415.773,170.632,35.172,156.614
C00540=1048.045,93.564,415.751,170.634,35.175,156.614
C00541=1048.051,93.849,415.729,170.636,35.177,156.615
C00542=1048.058,94.136,415.707,170.638,35.179,156.615
C00543=1048.064,94.385,415.689,170.639,35.180,156.615
C00544=1048.070,94.634,415.669,170.641,35.182,156.616
C00545=1048.077,94.883,415.650,170.643,35.184,156.616
C00546=1048.082,95.133,415.631,170.645,35.186,156.616
C00547=1048.089,95.382,415.612,170.647,35.187,156.617
C00548=1048.095,95.630,415.592,170.648,35.189,156.617
C00549=1048.101,95.880,415.573,170.650,35.191,156.617
C00550=1048.107,96.129,415.554,170.652,35.193,156.618
C00551=1048.114,96.379,415.535,170.653,35.194,156.618
C00552=1048.120,96.628,415.515,170.655,35.196,156.618
C00553=1048.126,96.877,415.497,170.657,35.198,156.619
C00554=1048.132,97.126,415.477,170.658,35.200,156.619
C00555=1048.138,97.376,415.458,170.661,35.201,156.619
C00556=1048.144,97.624,415.439,170.663,35.203,156.619
C00557=1048.150,97.874,415.419,170.664,35.205,156.620
C00558=1048.156,98.123,415.401,170.666,35.207,156.620
C00559=1048.162,98.371,415.381,170.668,35.209,156.620
C00560=1048.170,98.621,415.362,170.669,35.210,156.621
C00561=1048.175,98.871,415.343,170.671,35.212,156.621
C00562=1048.182,99.119,415.323,170.673,35.214,156.621
C00563=1048.188,99.369,415.304,170.675,35.216,156.622
C00564=1048.194,99.617,415.284,170.677,35.217,156.622
C00565=1048.200,99.867,415.265,170.678,35.219,156.622
C00566=1048.206,100.116,415.246,170.680,35.221,156.623
C00567=1048.213,100.365,415.226,170.682,35.223,156.623
C00568=1048.219,100.615,415.207,170.683,35.224,156.623
C00569=1048.224,100.864,415.188,170.685,35.226,156.624
C00570=1048.230,101.113,415.168,170.687,35.228,156.624
C00571=1048.237,101.362,415.149,170.689,35.230,156.624
C00572=1048.243,101.611,415.129,170.691,35.232,156.625
C00573=1048.249,101.860,415.110,170.693,35.234,156.625
C00574=1048.255,102.110,415.090,170.694,35.235,156.625
C00575=1048.261,102.359,415.071,170.696,35.237,156.625
C00576=1048.268,102.608,415.051,170.698,35.239,156.626
C00577=1048.273,102.857,415.032,170.699,35.241,156.626
C00578=1048.279,103.106,415.012,170.701,35.243,156.626
C00579=1048.285,103.355,414.993,170.704,35.245,156.627
C00580=1048.291,103.604,414.973,170.705,35.247,156.627
C00581=1048.298,103.854,414.954,170.707,35.249,156.628
C00582=1048.304,104.103,414.934,170.708,35.250,156.628
C00583=1048.310,104.352,414.914,170.710,35.252,156.628
C00584=1048.316,104.601,414.895,170.712,35.254,156.628
C00585=1048.322,104.850,414.875,170.713,35.256,156.629
C00586=1048.327,105.099,414.855,170.715,35.257,156.629
C00587=1048.335,105.349,414.836,170.718,35.259,156.629
C00588=1048.340,105.598,414.816,170.719,35.261,156.630
C00589=1048.346,105.847,414.796,170.721,35.263,156.630
C00590=1048.352,106.096,414.777,170.723,35.265,156.630
C00591=1048.358,106.345,414.757,170.724,35.266,156.631
C00592=1048.365,106.595,414.737,170.726,35.268,156.631
C00593=1048.371,106.843,414.718,170.728,35.270,156.631
C00594=1048.377,107.093,414.698,170.729,35.272,156.632
C00595=1048.383,107.341,414.678,170.732,35.273,156.632
C00596=1048.390,107.591,414.658,170.734,35.275,156.632
C00597=1048.395,107.840,414.639,170.735,35.277,156.633
C00598=1048.401,108.089,414.619,170.737,35.279,156.633
C00599=1048.407,108.338,414.599,170.739,35.281,156.633
C00600=1048.414,108.588,414.580,170.740,35.283,156.634
C00601=1048.420,108.837,414.560,170.742,35.284,156.634
C00602=1048.426,109.085,414.540,170.744,35.286,156.634
C00603=1048.433,109.371,414.517,170.747,35.289,156.635
C00604=1048.440,109.657,414.495,170.749,35.291,156.635
C00605=1048.447,109.943,414.472,170.751,35.292,156.635
C00606=1048.455,110.229,414.449,170.752,35.294,156.636
C00607=1048.461,110.478,414.429,170.754,35.296,156.636
C00608=1048.467,110.728,414.410,170.756,35.298,156.636
C00609=1048.473,110.977,414.390,170.758,35.300,156.637
C00610=1048.479,111.225,414.370,170.760,35.302,156.637
C00611=1048.485,111.475,414.350,170.762,35.304,156.637
C00612=1048.491,111.724,414.330,170.764,35.305,156.638
C00613=1048.497,111.973,414.310,170.765,35.307,156.638
C00614=1048.503,112.222,414.290,170.767,35.309,156.638
C00615=1048.510,112.471,414.270,170.769,35.311,156.639
C00616=1048.516,112.720,414.250,170.770,35.313,156.639
C00617=1048.522,112.969,414.230,170.772,35.315,156.639
C00618=1048.528,113.219,414.210,170.775,35.317,156.640
C00619=1048.534,113.467,414.190,170.776,35.318,156.640
C00620=1048.540,113.717,414.171,170.778,35.320,156.640
C00621=1048.547,113.966,414.150,170.780,35.322,156.641
C00622=1048.553,114.215,414.130,170.781,35.324,156.641
C00623=1048.558,114.464,414.110,170.783,35.326,156.641
C00624=1048.564,114.713,414.090,170.785,35.328,156.642
C00625=1048.570,114.963,414.070,170.787,35.330,156.642
C00626=1048.576,115.212,414.049,170.789,35.332,156.642
C00627=1048.582,115.461,414.029,170.791,35.334,156.643
C00628=1048.588,115.710,414.009,170.792,35.336,156.643
C00629=1048.594,115.959,413.989,170.794,35.337,156.643
C00630=1048.599,116.208,413.968,170.796,35.339,156.644
C00631=1048.605,116.457,413.948,170.797,35.341,156.644
C00632=1048.612,116.706,413.928,170.800,35.343,156.645
C00633=1048.618,116.955,413.908,170.802,35.345,156.645
C00634=1048.623,117.204,413.887,170.803,35.347,156.645
C00635=1048.630,117.454,413.867,170.805,35.349,156.646
C00636=1048.636,117.703,413.847,170.807,35.351,156.646
C00637=1048.641,117.952,413.827,170.808,35.353,156.646
C00638=1048.648,118.201,413.806,170.810,35.354,156.647
C00639=1048.654,118.450,413.786,170.813,35.356,156.647
C00640=1048.660,118.698,413.766,170.814,35.358,156.647
C00641=1048.666,118.948,413.745,170.816,35.360,156.648
C00642=1048.672,119.197,413.725,170.818,35.362,156.648
C00643=1048.679,119.446,413.704,170.820,35.363,156.648
C00644=1048.684,119.696,413.684,170.821,35.365,156.649
C00645=1048.690,119.944,413.664,170.823,35.367,156.649
C00646=1048.696,120.194,413.644,170.825,35.369,156.649
C00647=1048.702,120.443,413.624,170.827,35.371,156.650
C00648=1048.708,120.692,413.603,170.829,35.373,156.650
C00649=1048.715,120.941,413.582,170.831,35.375,156.650
C00650=1048.721,121.189,413.562,170.832,35.377,156.651
C00651=1048.726,121.439,413.541,170.834,35.378,156.651
C00652=1048.732,121.688,413.521,170.836,35.380,156.651
C00653=1048.738,121.937,413.501,170.838,35.382,156.652
C00654=1048.745,122.186,413.480,170.840,35.384,156.652
C00655=1048.751,122.435,413.460,170.842,35.386,156.652
C00656=1048.757,122.684,413.439,170.844,35.388,156.653
C00657=1048.762,122.934,413.419,170.845,35.390,156.653
C00658=1048.769,123.183,413.398,170.847,35.392,156.653
C00659=1048.775,123.431,413.378,170.849,35.394,156.654
C00660=1048.781,123.681,413.357,170.851,35.396,156.654
C00661=1048.787,123.930,413.337,170.853,35.397,156.654
C00662=1048.793,124.179,413.317,170.855,35.399,156.655
C00663=1048.799,124.428,413.295,170.857,35.401,156.655
C00664=1048.805,124.677,413.275,170.858,35.403,156.655
C00665=1048.812,124.926,413.255,170.860,35.405,156.656
C00666=1048.817,125.175,413.234,170.862,35.407,156.656
C00667=1048.825,125.462,413.210,170.864,35.409,156.656
C00668=1048.832,125.747,413.187,170.867,35.411,156.657
C00669=1048.839,126.032,413.163,170.869,35.413,156.657
C00670=1048.846,126.318,413.139,170.871,35.415,156.658
C00671=1048.852,126.567,413.119,170.873,35.417,156.658
C00672=1048.858,126.816,413.099,170.874,35.419,156.658
C00673=1048.864,127.065,413.078,170.876,35.421,156.659
C00674=1048.870,127.314,413.058,170.879,35.423,156.659
C00675=1048.876,127.564,413.037,170.881,35.425,156.659
C00676=1048.883,127.812,413.016,170.882,35.426,156.660
C00677=1048.889,128.062,412.996,170.884,35.428,156.660
C00678=1048.895,128.310,412.974,170.886,35.430,156.660
C00679=1048.901,128.560,412.954,170.888,35.432,156.661
C00680=1048.908,128.809,412.934,170.889,35.434,156.661
C00681=1048.914,129.058,412.912,170.892,35.436,156.661
C00682=1048.920,129.307,412.892,170.894,35.437,156.662
C00683=1048.926,129.555,412.871,170.896,35.439,156.662
C00684=1048.932,129.805,412.851,170.897,35.441,156.662
C00685=1048.938,130.054,412.831,170.899,35.443,156.663
C00686=1048.944,130.303,412.809,170.901,35.445,156.663
C00687=1048.951,130.553,412.789,170.903,35.447,156.663
C00688=1048.957,130.801,412.768,170.905,35.449,156.664
C00689=1048.963,131.051,412.747,170.907,35.450,156.664
C00690=1048.970,131.299,412.726,170.909,35.452,156.664
C00691=1048.975,131.549,412.705,170.911,35.454,156.665
C00692=1048.982,131.798,412.684,170.912,35.456,156.665
C00693=1048.988,132.047,412.664,170.914,35.458,156.665
C00694=1048.994,132.296,412.642,170.916,35.460,156.666
C00695=1049.000,132.544,412.622,170.919,35.462,156.666
C00696=1049.006,132.794,412.601,170.920,35.464,156.666
C00697=1049.011,133.042,412.579,170.922,35.466,156.667
C00698=1049.018,133.292,412.559,170.924,35.467,156.667
C00699=1049.024,133.541,412.537,170.926,35.469,156.667
C00700=1049.030,133.790,412.516,170.927,35.471,156.668
C00701=1049.036,134.039,412.496,170.929,35.474,156.668
C00702=1049.042,134.288,412.474,170.932,35.476,156.669
C00703=1049.048,134.537,412.453,170.934,35.477,156.669
C00704=1049.054,134.786,412.433,170.935,35.479,156.669
C00705=1049.060,135.035,412.411,170.937,35.481,156.670
C00706=1049.066,135.284,412.390,170.939,35.483,156.670
C00707=1049.072,135.533,412.370,170.941,35.485,156.670
C00708=1049.079,135.782,412.348,170.944,35.487,156.671
C00709=1049.085,136.031,412.326,170.945,35.489,156.671
C00710=1049.091,136.280,412.306,170.947,35.491,156.671
C00711=1049.097,136.529,412.285,170.949,35.493,156.672
C00712=1049.102,136.778,412.264,170.951,35.494,156.672
C00713=1049.109,137.027,412.242,170.952,35.496,156.672
C00714=1049.115,137.277,412.222,170.954,35.498,156.673
C00715=1049.121,137.525,412.200,170.957,35.500,156.673
C00716=1049.127,137.774,412.179,170.959,35.502,156.674
C00717=1049.133,138.024,412.157,170.961,35.504,156.674
C00718=1049.139,138.272,412.137,170.962,35.506,156.674
C00719=1049.145,138.522,412.115,170.964,35.508,156.675
C00720=1049.151,138.771,412.094,170.966,35.510,156.675
C00721=1049.157,139.019,412.073,170.969,35.512,156.675
C00722=1049.164,139.268,412.051,170.970,35.514,156.676
C00723=1049.170,139.518,412.031,170.972,35.516,156.676
C00724=1049.175,139.766,412.009,170.974,35.518,156.676
C00725=1049.181,140.016,411.988,170.976,35.520,156.677
C00726=1049.188,140.265,411.966,170.978,35.521,156.677
C00727=1049.193,140.513,411.945,170.979,35.524,156.678
C00728=1049.199,140.763,411.923,170.982,35.526,156.678
C00729=1049.205,141.012,411.901,170.984,35.528,156.678
C00730=1049.212,141.260,411.881,170.986,35.530,156.679
C00731=1049.219,141.546,411.856,170.988,35.532,156.679
C00732=1049.225,141.831,411.831,170.990,35.534,156.679
C00733=1049.232,142.117,411.808,170.993,35.536,156.680
C00734=1049.239,142.403,411.782,170.995,35.539,156.680
C00735=1049.246,142.652,411.761,170.997,35.541,156.681
C00736=1049.251,142.900,411.739,170.999,35.543,156.681
C00737=1049.257,143.150,411.718,171.000,35.545,156.681
C00738=1049.263,143.399,411.696,171.002,35.546,156.682
C00739=1049.269,143.647,411.675,171.004,35.548,156.682
C00740=1049.275,143.896,411.653,171.007,35.550,156.682
C00741=1049.281,144.146,411.632,171.009,35.553,156.683
C00742=1049.287,144.395,411.610,171.010,35.555,156.683
C00743=1049.293,144.643,411.589,171.012,35.557,156.684
C00744=1049.299,144.893,411.567,171.014,35.558,156.684
C00745=1049.305,145.142,411.545,171.016,35.560,156.684
C00746=1049.312,145.391,411.524,171.019,35.562,156.685
C00747=1049.318,145.639,411.503,171.021,35.564,156.685
C00748=1049.324,145.888,411.481,171.022,35.567,156.685
C00749=1049.330,146.138,411.460,171.024,35.568,156.686
C00750=1049.336,146.387,411.438,171.026,35.570,156.686
C00751=1049.343,146.635,411.416,171.028,35.572,156.687
C00752=1049.348,146.884,411.395,171.031,35.574,156.687
C00753=1049.355,147.133,411.373,171.033,35.576,156.687
C00754=1049.361,147.382,411.351,171.034,35.578,156.688
C00755=1049.367,147.632,411.330,171.036,35.580,156.688
C00756=1049.373,147.881,411.308,171.038,35.582,156.688
C00757=1049.378,148.130,411.286,171.040,35.584,156.689
C00758=1049.384,148.378,411.264,171.043,35.586,156.689
C00759=1049.390,148.627,411.242,171.045,35.588,156.689
C00760=1049.397,148.877,411.220,171.046,35.590,156.690
C00761=1049.403,149.126,411.199,171.048,35.592,156.690
C00762=1049.408,149.374,411.178,171.050,35.594,156.691
C00763=1049.415,149.623,411.155,171.052,35.596,156.691
C00764=1049.421,149.872,411.134,171.055,35.598,156.691
C00765=1049.426,150.122,411.111,171.057,35.600,156.692
C00766=1049.433,150.371,411.090,171.058,35.602,156.692
C00767=1049.438,150.619,411.068,171.060,35.604,156.692
C00768=1049.445,150.868,411.046,171.062,35.607,156.693
C00769=1049.451,151.117,411.024,171.064,35.608,156.693
C00770=1049.456,151.366,411.002,171.067,35.610,156.694
C00771=1049.463,151.615,410.980,171.069,35.612,156.694
C00772=1049.469,151.864,410.958,171.071,35.615,156.694
C00773=1049.475,152.113,410.936,171.072,35.617,156.695
C00774=1049.481,152.361,410.915,171.074,35.618,156.695
C00775=1049.486,152.611,410.892,171.076,35.620,156.696
C00776=1049.493,152.860,410.870,171.079,35.623,156.696
C00777=1049.499,153.109,410.848,171.081,35.625,156.696
C00778=1049.505,153.358,410.827,171.083,35.627,156.697
C00779=1049.511,153.607,410.804,171.085,35.628,156.697
C00780=1049.517,153.856,410.782,171.087,35.631,156.698
C00781=1049.523,154.105,410.760,171.089,35.633,156.698
C00782=1049.529,154.353,410.739,171.091,35.635,156.698
C00783=1049.534,154.603,410.716,171.093,35.636,156.699
C00784=1049.541,154.851,410.694,171.095,35.639,156.699
C00785=1049.547,155.100,410.672,171.097,35.641,156.699
C00786=1049.554,155.349,410.650,171.099,35.643,156.700
C00787=1049.559,155.599,410.628,171.102,35.645,156.700
C00788=1049.565,155.847,410.605,171.104,35.647,156.701
C00789=1049.571,156.097,410.583,171.105,35.649,156.701
C00790=1049.577,156.345,410.561,171.107,35.651,156.701
C00791=1049.583,156.594,410.539,171.109,35.653,156.702
C00792=1049.589,156.843,410.516,171.111,35.655,156.702
C00793=1049.595,157.092,410.495,171.114,35.657,156.702
C00794=1049.601,157.340,410.473,171.116,35.660,156.703
C00795=1049.608,157.626,410.447,171.118,35.661,156.703
C00796=1049.615,157.911,410.421,171.120,35.664,156.704
C00797=1049.622,158.197,410.396,171.122,35.666,156.704
C00798=1049.629,158.481,410.370,171.126,35.669,156.705
C00799=1049.635,158.730,410.348,171.127,35.671,156.705
C00800=1049.641,158.979,410.325,171.129,35.673,156.705
C00801=1049.647,159.229,410.304,171.131,35.675,156.706
C00802=1049.653,159.477,410.281,171.133,35.677,156.706
C00803=1049.659,159.726,410.259,171.136,35.679,156.707
C00804=1049.665,159.975,410.237,171.138,35.681,156.707
C00805=1049.672,160.224,410.215,171.140,35.683,156.707
C00806=1049.677,160.473,410.192,171.142,35.685,156.708
C00807=1049.683,160.722,410.170,171.144,35.688,156.708
C00808=1049.689,160.971,410.147,171.146,35.689,156.709
C00809=1049.695,161.220,410.124,171.149,35.692,156.709
C00810=1049.701,161.469,410.101,171.150,35.694,156.709
C00811=1049.706,161.718,410.079,171.152,35.696,156.710
C00812=1049.712,161.967,410.057,171.154,35.698,156.710
C00813=1049.718,162.216,410.034,171.156,35.701,156.711
C00814=1049.724,162.465,410.011,171.159,35.702,156.711
C00815=1049.729,162.714,409.988,171.161,35.705,156.711
C00816=1049.736,162.963,409.966,171.163,35.707,156.712
C00817=1049.742,163.212,409.943,171.165,35.709,156.712
C00818=1049.747,163.460,409.920,171.167,35.711,156.713
C00819=1049.753,163.709,409.897,171.170,35.714,156.713
C00820=1049.759,163.957,409.875,171.171,35.716,156.714
C00821=1049.765,164.206,409.852,171.173,35.718,156.714
C00822=1049.770,164.456,409.830,171.175,35.720,156.714
C00823=1049.776,164.705,409.807,171.177,35.722,156.715
C00824=1049.782,164.953,409.784,171.180,35.725,156.715
C00825=1049.788,165.202,409.762,171.182,35.727,156.716
C00826=1049.794,165.451,409.739,171.184,35.729,156.716
C00827=1049.799,165.700,409.716,171.186,35.731,156.716
C00828=1049.806,165.949,409.693,171.188,35.733,156.717
C00829=1049.812,166.198,409.670,171.191,35.735,156.717
C00830=1049.818,166.447,409.647,171.193,35.738,156.718
C00831=1049.824,166.696,409.624,171.195,35.740,156.718
C00832=1049.829,166.945,409.601,171.197,35.742,156.719
C00833=1049.835,167.194,409.578,171.199,35.744,156.719
C00834=1049.841,167.442,409.556,171.202,35.746,156.719
C00835=1049.847,167.691,409.533,171.203,35.748,156.720
C00836=1049.853,167.940,409.510,171.205,35.751,156.720
C00837=1049.859,168.189,409.487,171.207,35.753,156.721
C00838=1049.865,168.438,409.464,171.209,35.755,156.721
C00839=1049.870,168.687,409.441,171.212,35.757,156.721
C00840=1049.877,168.935,409.419,171.214,35.759,156.722
C00841=1049.882,169.184,409.396,171.216,35.762,156.722
C00842=1049.888,169.433,409.373,171.218,35.764,156.723
C00843=1049.895,169.683,409.350,171.220,35.766,156.723
C00844=1049.900,169.932,409.327,171.223,35.768,156.724
C00845=1049.906,170.180,409.304,171.225,35.771,156.724
C00846=1049.912,170.429,409.282,171.227,35.772,156.724
C00847=1049.918,170.678,409.259,171.229,35.775,156.725
C00848=1049.924,170.926,409.235,171.231,35.777,156.725
C00849=1049.930,171.175,409.212,171.234,35.779,156.726
C00850=1049.936,171.425,409.189,171.236,35.781,156.726
C00851=1049.942,171.674,409.166,171.238,35.784,156.726
C00852=1049.949,171.922,409.143,171.240,35.785,156.727
C00853=1049.954,172.171,409.121,171.242,35.788,156.727
C00854=1049.960,172.419,409.097,171.245,35.790,156.728
C00855=1049.966,172.668,409.074,171.247,35.792,156.728
C00856=1049.972,172.918,409.051,171.249,35.795,156.729
C00857=1049.978,173.167,409.028,171.251,35.797,156.729
C00858=1049.984,173.416,409.005,171.253,35.799,156.729
C00859=1049.991,173.699,408.978,171.256,35.802,156.730
C00860=1049.998,173.985,408.952,171.259,35.804,156.730
C00861=1050.005,174.269,408.925,171.261,35.807,156.731
C00862=1050.012,174.554,408.899,171.263,35.809,156.731
C00863=1050.017,174.803,408.876,171.265,35.811,156.732
C00864=1050.024,175.052,408.853,171.268,35.813,156.732
C00865=1050.031,175.301,408.829,171.270,35.816,156.733
C00866=1050.036,175.550,408.806,171.272,35.818,156.733
C00867=1050.042,175.798,408.783,171.274,35.820,156.733
C00868=1050.048,176.047,408.760,171.277,35.822,156.734
C00869=1050.054,176.296,408.736,171.280,35.824,156.734
C00870=1050.060,176.545,408.713,171.282,35.826,156.735
C00871=1050.066,176.794,408.690,171.284,35.829,156.735
C00872=1050.072,177.042,408.667,171.286,35.831,156.735
C00873=1050.079,177.292,408.644,171.289,35.833,156.736
C00874=1050.085,177.540,408.620,171.291,35.836,156.736
C00875=1050.091,177.789,408.598,171.293,35.837,156.737
C00876=1050.097,178.038,408.574,171.295,35.840,156.737
C00877=1050.103,178.287,408.551,171.297,35.842,156.738
C00878=1050.109,178.536,408.528,171.300,35.844,156.738
C00879=1050.115,178.785,408.504,171.302,35.846,156.738
C00880=1050.121,179.034,408.481,171.304,35.849,156.739
C00881=1050.127,179.282,408.457,171.306,35.850,156.739
C00882=1050.134,179.531,408.434,171.308,35.853,156.740
C00883=1050.140,179.779,408.411,171.311,35.855,156.740
C00884=1050.146,180.028,408.388,171.313,35.857,156.741
C00885=1050.153,180.277,408.364,171.316,35.860,156.741
C00886=1050.158,180.526,408.341,171.318,35.861,156.741
C00887=1050.165,180.775,408.317,171.320,35.864,156.742
C00888=1050.171,181.024,408.294,171.323,35.866,156.742
C00889=1050.177,181.272,408.270,171.325,35.868,156.743
C00890=1050.183,181.522,408.247,171.327,35.871,156.743
C00891=1050.189,181.770,408.223,171.329,35.873,156.744
C00892=1050.196,182.020,408.200,171.332,35.875,156.744
C00893=1050.202,182.268,408.176,171.334,35.877,156.744
C00894=1050.208,182.516,408.152,171.336,35.879,156.745
C00895=1050.214,182.766,408.129,171.339,35.882,156.745
C00896=1050.220,183.014,408.105,171.341,35.884,156.746
C00897=1050.226,183.264,408.082,171.344,35.886,156.746
C00898=1050.233,183.512,408.059,171.346,35.888,156.747
C00899=1050.240,183.761,408.035,171.348,35.890,156.747
C00900=1050.245,184.010,408.012,171.350,35.893,156.748
C00901=1050.251,184.258,407.988,171.352,35.895,156.748
C00902=1050.257,184.507,407.964,171.355,35.897,156.748
C00903=1050.262,184.756,407.940,171.357,35.900,156.749
C00904=1050.268,185.005,407.917,171.359,35.902,156.749
C00905=1050.274,185.254,407.892,171.361,35.905,156.750
C00906=1050.280,185.502,407.868,171.365,35.907,156.750
C00907=1050.286,185.751,407.844,171.367,35.909,156.751
C00908=1050.292,186.000,407.821,171.369,35.912,156.751
C00909=1050.298,186.249,407.797,171.371,35.914,156.752
C00910=1050.304,186.498,407.773,171.374,35.916,156.752
C00911=1050.310,186.746,407.749,171.376,35.919,156.753
C00912=1050.315,186.995,407.725,171.378,35.921,156.753
C00913=1050.322,187.244,407.701,171.380,35.924,156.753
C00914=1050.327,187.492,407.676,171.383,35.926,156.754
C00915=1050.333,187.741,407.653,171.385,35.929,156.754
C00916=1050.339,187.991,407.629,171.388,35.931,156.755
C00917=1050.345,188.239,407.605,171.390,35.933,156.755
C00918=1050.351,188.488,407.580,171.392,35.936,156.756
C00919=1050.357,188.736,407.557,171.395,35.938,156.756
C00920=1050.363,188.986,407.532,171.397,35.941,156.757
C00921=1050.369,189.234,407.509,171.399,35.943,156.757
C00922=1050.374,189.483,407.484,171.401,35.945,156.758
C00923=1050.381,189.767,407.457,171.405,35.948,156.758
C00924=1050.388,190.052,407.429,171.407,35.951,156.759
C00925=1050.395,190.336,407.402,171.410,35.954,156.759
C00926=1050.402,190.620,407.374,171.413,35.956,156.760
C00927=1050.408,190.869,407.350,171.415,35.959,156.760
C00928=1050.414,191.118,407.325,171.417,35.961,156.761
C00929=1050.419,191.366,407.301,171.420,35.963,156.761
C00930=1050.426,191.615,407.277,171.422,35.966,156.762
C00931=1050.431,191.864,407.253,171.425,35.968,156.762
C00932=1050.438,192.113,407.229,171.427,35.971,156.763
C00933=1050.443,192.361,407.205,171.429,35.973,156.763
C00934=1050.450,192.610,407.181,171.431,35.976,156.764
C00935=1050.455,192.859,407.156,171.435,35.978,156.764
C00936=1050.462,193.108,407.132,171.437,35.981,156.765
C00937=1050.467,193.356,407.108,171.439,35.983,156.765
C00938=1050.474,193.605,407.083,171.441,35.986,156.766
C00939=1050.479,193.853,407.059,171.444,35.988,156.766
C00940=1050.485,194.103,407.034,171.446,35.990,156.767
C00941=1050.492,194.352,407.010,171.449,35.993,156.767
C00942=1050.497,194.600,406.986,171.451,35.995,156.768
C00943=1050.504,194.849,406.962,171.454,35.998,156.768
C00944=1050.510,195.097,406.937,171.456,36.000,156.769
C00945=1050.516,195.346,406.913,171.458,36.002,156.769
C00946=1050.522,195.595,406.889,171.461,36.005,156.769
C00947=1050.528,195.844,406.865,171.464,36.007,156.770
C00948=1050.534,196.092,406.840,171.466,36.009,156.770
C00949=1050.540,196.341,406.816,171.468,36.012,156.771
C00950=1050.546,196.590,406.791,171.470,36.014,156.771
C00951=1050.552,196.839,406.767,171.474,36.017,156.772
C00952=1050.558,197.087,406.742,171.476,36.019,156.772
C00953=1050.564,197.336,406.718,171.478,36.022,156.773
C00954=1050.571,197.585,406.694,171.480,36.024,156.773
C00955=1050.577,197.833,406.669,171.484,36.027,156.774
C00956=1050.583,198.082,406.645,171.486,36.029,156.774
C00957=1050.589,198.331,406.620,171.488,36.031,156.775
C00958=1050.595,198.579,406.595,171.490,36.034,156.775
C00959=1050.601,198.828,406.571,171.494,36.036,156.776
C00960=1050.607,199.078,406.546,171.496,36.039,156.776
C00961=1050.614,199.325,406.522,171.498,36.042,156.777
C00962=1050.620,199.575,406.497,171.500,36.044,156.777
C00963=1050.625,199.824,406.473,171.504,36.047,156.778
C00964=1050.632,200.072,406.448,171.506,36.049,156.778
C00965=1050.638,200.321,406.424,171.508,36.052,156.779
C00966=1050.645,200.569,406.399,171.510,36.054,156.779
C00967=1050.651,200.818,406.374,171.514,36.056,156.780
C00968=1050.657,201.067,406.349,171.516,36.059,156.780
C00969=1050.663,201.315,406.325,171.518,36.061,156.781
C00970=1050.669,201.564,406.300,171.520,36.064,156.781
C00971=1050.675,201.813,406.275,171.524,36.066,156.782
C00972=1050.681,202.062,406.250,171.526,36.069,156.782
C00973=1050.687,202.310,406.226,171.528,36.072,156.783
C00974=1050.693,202.559,406.201,171.531,36.074,156.783
C00975=1050.699,202.808,406.176,171.534,36.077,156.784
C00976=1050.705,203.056,406.151,171.536,36.079,156.784
C00977=1050.711,203.305,406.126,171.538,36.081,156.785
C00978=1050.717,203.554,406.102,171.541,36.084,156.785
C00979=1050.723,203.803,406.076,171.544,36.087,156.786
C00980=1050.729,204.051,406.051,171.546,36.089,156.786
C00981=1050.735,204.300,406.027,171.548,36.092,156.787
C00982=1050.741,204.549,406.001,171.552,36.095,156.787
C00983=1050.747,204.797,405.976,171.554,36.097,156.788
C00984=1050.752,205.046,405.952,171.556,36.100,156.788
C00985=1050.759,205.294,405.927,171.559,36.103,156.789
C00986=1050.766,205.543,405.902,171.562,36.105,156.789
C00987=1050.790,206.596,405.796,171.789,36.201,156.808
C00988=1050.797,206.846,405.769,171.790,36.205,156.809
C00989=1050.804,207.098,405.743,171.793,36.208,156.809
C00990=1050.810,207.349,405.717,171.795,36.211,156.810
C00991=1050.817,207.600,405.691,171.797,36.215,156.811
C00992=1050.824,207.849,405.664,171.799,36.218,156.812
C00993=1050.829,208.098,405.638,171.801,36.221,156.812
C00994=1050.836,208.346,405.612,171.803,36.225,156.813
C00995=1050.843,208.594,405.586,171.805,36.228,156.814
C00996=1050.849,208.843,405.559,171.806,36.232,156.814
C00997=1050.855,209.092,405.534,171.809,36.235,156.815
C00998=1050.862,209.340,405.507,171.811,36.238,156.816
C00999=1050.869,209.588,405.481,171.813,36.242,156.816
C01000=1050.874,209.837,405.455,171.815,36.245,156.817
C01001=1050.881,210.086,405.429,171.816,36.248,156.818
C01002=1050.888,210.334,405.403,171.819,36.252,156.819
C01003=1050.893,210.582,405.376,171.821,36.256,156.819
C01004=1050.901,210.831,405.350,171.823,36.259,156.820
C01005=1050.906,211.080,405.324,171.825,36.262,156.821
C01006=1050.913,211.329,405.298,171.827,36.266,156.821
C01007=1050.920,211.577,405.272,171.829,36.269,156.822
C01008=1050.925,211.825,405.245,171.831,36.272,156.823
C01009=1050.933,212.074,405.218,171.832,36.275,156.823
C01010=1050.938,212.322,405.192,171.835,36.279,156.824
C01011=1050.945,212.570,405.166,171.837,36.283,156.825
C01012=1050.951,212.820,405.139,171.839,36.286,156.825
C01013=1050.957,213.068,405.113,171.841,36.289,156.826
C01014=1050.964,213.317,405.086,171.843,36.293,156.827
C01015=1050.970,213.565,405.060,171.845,36.296,156.828
C01016=1050.976,213.814,405.034,171.847,36.299,156.828
C01017=1050.983,214.062,405.007,171.850,36.303,156.829
C01018=1050.989,214.311,404.981,171.851,36.306,156.830
C01019=1050.996,214.560,404.954,171.853,36.310,156.830
C01020=1051.002,214.808,404.928,171.856,36.313,156.831
C01021=1051.008,215.056,404.901,171.857,36.316,156.832
C01022=1051.015,215.305,404.874,171.860,36.320,156.832
C01023=1051.021,215.553,404.848,171.862,36.323,156.833
C01024=1051.028,215.802,404.821,171.863,36.326,156.834
C01025=1051.033,216.050,404.795,171.866,36.330,156.835
C01026=1051.041,216.299,404.768,171.868,36.333,156.835
C01027=1051.046,216.548,404.742,171.870,36.337,156.836
C01028=1051.053,216.796,404.714,171.872,36.340,156.837
C01029=1051.059,217.044,404.688,171.874,36.343,156.837
C01030=1051.066,217.293,404.661,171.877,36.347,156.838
C01031=1051.072,217.541,404.635,171.878,36.350,156.839
C01032=1051.079,217.790,404.608,171.881,36.353,156.839
C01033=1051.085,218.038,404.582,171.883,36.357,156.840
C01034=1051.092,218.287,404.555,171.884,36.360,156.841
C01035=1051.097,218.536,404.528,171.887,36.364,156.842
C01036=1051.105,218.784,404.501,171.889,36.366,156.842
C01037=1051.111,219.032,404.474,171.891,36.370,156.843
C01038=1051.118,219.281,404.448,171.893,36.373,156.844
C01039=1051.123,219.529,404.421,171.895,36.377,156.844
C01040=1051.130,219.778,404.394,171.898,36.380,156.845
C01041=1051.136,220.026,404.368,171.899,36.383,156.846
C01042=1051.143,220.275,404.340,171.902,36.387,156.846
C01043=1051.150,220.523,404.314,171.904,36.390,156.847
C01044=1051.156,220.780,404.286,171.906,36.393,156.848
C01045=1051.163,221.037,404.258,171.908,36.397,156.848
C01046=1051.169,221.294,404.231,171.910,36.400,156.849
C01047=1051.176,221.550,404.203,171.913,36.404,156.850
C01048=1051.182,221.798,404.176,171.915,36.407,156.851
C01049=1051.189,222.047,404.149,171.917,36.410,156.851
C01050=1051.194,222.296,404.122,171.919,36.414,156.852
C01051=1051.201,222.544,404.094,171.921,36.417,156.853
C01052=1051.207,222.792,404.068,171.924,36.420,156.853
C01053=1051.213,223.041,404.041,171.926,36.424,156.854
C01054=1051.221,223.290,404.014,171.927,36.427,156.855
C01055=1051.226,223.538,403.987,171.930,36.430,156.855
C01056=1051.233,223.786,403.959,171.932,36.434,156.856
C01057=1051.239,224.035,403.933,171.935,36.437,156.857
C01058=1051.245,224.283,403.905,171.936,36.441,156.858
C01059=1051.252,224.532,403.878,171.938,36.444,156.858
C01060=1051.258,224.780,403.852,171.941,36.447,156.859
C01061=1051.265,225.029,403.824,171.943,36.451,156.860
C01062=1051.271,225.277,403.797,171.945,36.454,156.860
C01063=1051.278,225.526,403.770,171.947,36.457,156.861
C01064=1051.284,225.775,403.743,171.949,36.460,156.862
C01065=1051.290,226.022,403.715,171.952,36.464,156.862
C01066=1051.296,226.271,403.688,171.954,36.467,156.863
C01067=1051.303,226.520,403.661,171.956,36.470,156.864
C01068=1051.310,226.768,403.634,171.958,36.473,156.864
C01069=1051.316,227.016,403.607,171.961,36.477,156.865
C01070=1051.323,227.265,403.579,171.963,36.480,156.866
C01071=1051.329,227.513,403.552,171.965,36.484,156.867
C01072=1051.335,227.762,403.525,171.968,36.487,156.867
C01073=1051.342,228.011,403.498,171.969,36.490,156.868
C01074=1051.348,228.258,403.470,171.972,36.493,156.869
C01075=1051.354,228.507,403.443,171.974,36.497,156.869
C01076=1051.361,228.756,403.416,171.976,36.500,156.870
C01077=1051.368,229.004,403.388,171.979,36.503,156.871
C01078=1051.373,229.253,403.361,171.980,36.506,156.871
C01079=1051.380,229.501,403.333,171.983,36.510,156.872
C01080=1051.387,229.750,403.306,171.985,36.513,156.873
C01081=1051.393,229.997,403.278,171.987,36.516,156.873
C01082=1051.399,230.246,403.251,171.990,36.520,156.874
C01083=1051.406,230.495,403.224,171.992,36.523,156.875
C01084=1051.412,230.743,403.196,171.994,36.526,156.875
C01085=1051.419,230.991,403.168,171.996,36.529,156.876
C01086=1051.425,231.240,403.141,171.999,36.533,156.877
C01087=1051.430,231.488,403.114,172.001,36.536,156.877
C01088=1051.437,231.737,403.086,172.003,36.540,156.878
C01089=1051.444,231.985,403.058,172.006,36.543,156.879
C01090=1051.450,232.233,403.030,172.008,36.546,156.880
C01091=1051.456,232.482,403.004,172.010,36.550,156.880
C01092=1051.463,232.730,402.976,172.012,36.553,156.881
C01093=1051.469,232.979,402.948,172.014,36.556,156.882
C01094=1051.475,233.227,402.920,172.017,36.559,156.882
C01095=1051.481,233.475,402.893,172.019,36.563,156.883
C01096=1051.488,233.724,402.865,172.022,36.566,156.884
C01097=1051.495,233.972,402.837,172.024,36.569,156.885
C01098=1051.501,234.221,402.809,172.027,36.573,156.885
C01099=1051.507,234.469,402.781,172.028,36.576,156.886
C01100=1051.514,234.718,402.754,172.030,36.579,156.887
C01101=1051.520,234.967,402.726,172.033,36.582,156.887
C01102=1051.526,235.216,402.699,172.035,36.586,156.888
C01103=1051.533,235.466,402.670,172.038,36.589,156.889
C01104=1051.539,235.714,402.642,172.040,36.592,156.889
C01105=1051.545,235.962,402.614,172.043,36.596,156.890
C01106=1051.551,236.211,402.587,172.045,36.599,156.891
C01107=1051.558,236.459,402.559,172.047,36.603,156.892
C01108=1051.565,236.707,402.531,172.049,36.606,156.892
C01109=1051.571,236.956,402.503,172.051,36.609,156.893
C01110=1051.577,237.205,402.475,172.054,36.612,156.894
C01111=1051.583,237.452,402.448,172.056,36.616,156.894
C01112=1051.589,237.701,402.419,172.058,36.619,156.895
C01113=1051.596,237.950,402.392,172.061,36.622,156.896
C01114=1051.603,238.198,402.364,172.063,36.625,156.896
C01115=1051.609,238.446,402.336,172.066,36.629,156.897
C01116=1051.616,238.695,402.307,172.068,36.632,156.898
C01117=1051.622,238.943,402.279,172.071,36.635,156.898
C01118=1051.628,239.191,402.252,172.073,36.638,156.899
C01119=1051.634,239.439,402.224,172.075,36.642,156.900
C01120=1051.641,239.688,402.196,172.078,36.645,156.900
C01121=1051.648,239.936,402.168,172.080,36.648,156.901
C01122=1051.654,240.185,402.139,172.083,36.651,156.902
C01123=1051.661,240.433,402.111,172.085,36.655,156.903
C01124=1051.667,240.682,402.083,172.088,36.658,156.903
C01125=1051.673,240.930,402.055,172.089,36.661,156.904
C01126=1051.680,241.178,402.027,172.091,36.664,156.905
C01127=1051.686,241.427,401.999,172.094,36.668,156.905
C01128=1051.693,241.675,401.971,172.096,36.671,156.906
C01129=1051.698,241.923,401.943,172.099,36.674,156.907
C01130=1051.705,242.171,401.915,172.101,36.677,156.907
C01131=1051.711,242.420,401.886,172.104,36.681,156.908
C01132=1051.718,242.668,401.858,172.106,36.684,156.909
C01133=1051.724,242.916,401.829,172.108,36.687,156.910
C01134=1051.730,243.165,401.801,172.111,36.691,156.910
C01135=1051.737,243.413,401.773,172.113,36.694,156.911
C01136=1051.743,243.662,401.744,172.116,36.697,156.912
C01137=1051.750,243.910,401.717,172.118,36.700,156.912
C01138=1051.756,244.158,401.688,172.121,36.704,156.913
C01139=1051.763,244.407,401.660,172.123,36.707,156.914
C01140=1051.769,244.655,401.631,172.126,36.710,156.914
C01141=1051.775,244.904,401.602,172.128,36.714,156.915
C01142=1051.782,245.151,401.574,172.130,36.717,156.916
C01143=1051.788,245.400,401.546,172.133,36.720,156.917
C01144=1051.794,245.648,401.517,172.135,36.723,156.917
C01145=1051.801,245.897,401.489,172.138,36.727,156.918
C01146=1051.807,246.145,401.460,172.140,36.730,156.919
C01147=1051.812,246.393,401.432,172.143,36.733,156.919
C01148=1051.819,246.641,401.403,172.145,36.737,156.920
C01149=1051.826,246.889,401.374,172.147,36.740,156.921
C01150=1051.831,247.138,401.346,172.150,36.743,156.922
C01151=1051.838,247.386,401.317,172.152,36.747,156.922
C01152=1051.844,247.634,401.289,172.155,36.750,156.923
C01153=1051.850,247.883,401.260,172.157,36.754,156.924
C01154=1051.856,248.131,401.231,172.160,36.757,156.924
C01155=1051.862,248.380,401.202,172.162,36.760,156.925
C01156=1051.868,248.625,401.174,172.165,36.764,156.926
C01157=1051.875,248.870,401.145,172.167,36.767,156.926
C01158=1051.881,249.116,401.117,172.170,36.770,156.927
C01159=1051.888,249.362,401.088,172.172,36.773,156.928
C01160=1051.894,249.608,401.060,172.174,36.777,156.929
C01161=1051.900,249.854,401.031,172.177,36.780,156.929
C01162=1051.906,250.100,401.003,172.179,36.783,156.930
C01163=1051.913,250.345,400.974,172.182,36.787,156.931
C01164=1051.919,250.594,400.945,172.184,36.790,156.931
C01165=1051.925,250.842,400.916,172.188,36.793,156.932
C01166=1051.931,251.090,400.888,172.190,36.796,156.933
C01167=1051.937,251.339,400.859,172.193,36.800,156.934
C01168=1051.943,251.587,400.830,172.195,36.803,156.934
C01169=1051.950,251.834,400.801,172.197,36.806,156.935
C01170=1051.957,252.083,400.772,172.200,36.810,156.936
C01171=1051.964,252.331,400.743,172.202,36.813,156.936
C01172=1051.970,252.580,400.714,172.205,36.816,156.937
C01173=1051.976,252.828,400.686,172.207,36.819,156.938
C01174=1051.982,253.076,400.657,172.210,36.823,156.938
C01175=1051.988,253.325,400.628,172.212,36.826,156.939
C01176=1051.994,253.573,400.599,172.215,36.829,156.940
C01177=1052.001,253.821,400.570,172.218,36.833,156.941
C01178=1052.007,254.069,400.540,172.221,36.835,156.941
C01179=1052.015,254.318,400.512,172.223,36.839,156.942
C01180=1052.021,254.566,400.483,172.225,36.842,156.943
C01181=1052.027,254.814,400.454,172.228,36.845,156.943
C01182=1052.033,255.062,400.425,172.230,36.849,156.944
C01183=1052.040,255.310,400.396,172.233,36.852,156.945
C01184=1052.046,255.558,400.366,172.235,36.855,156.946
C01185=1052.053,255.807,400.337,172.239,36.858,156.946
C01186=1052.059,256.055,400.308,172.241,36.862,156.947
C01187=1052.065,256.303,400.279,172.244,36.865,156.948
C01188=1052.071,256.551,400.250,172.246,36.868,156.948
C01189=1052.078,256.800,400.221,172.249,36.871,156.949
C01190=1052.085,257.048,400.191,172.251,36.875,156.950
C01191=1052.091,257.297,400.162,172.253,36.878,156.950
C01192=1052.098,257.544,400.133,172.257,36.881,156.951
C01193=1052.104,257.792,400.104,172.259,36.884,156.952
C01194=1052.111,258.041,400.075,172.262,36.888,156.953
C01195=1052.117,258.289,400.046,172.264,36.891,156.953
C01196=1052.124,258.537,400.017,172.267,36.894,156.954
C01197=1052.131,258.786,399.987,172.269,36.898,156.955
C01198=1052.137,259.034,399.958,172.273,36.901,156.955
C01199=1052.143,259.281,399.929,172.275,36.904,156.956
C01200=1052.150,259.530,399.900,172.278,36.907,156.957
C01201=1052.156,259.778,399.870,172.280,36.911,156.958
C01202=1052.163,260.026,399.841,172.283,36.914,156.958
C01203=1052.169,260.274,399.811,172.286,36.917,156.959
C01204=1052.176,260.523,399.782,172.288,36.920,156.960
C01205=1052.182,260.771,399.753,172.291,36.924,156.960
C01206=1052.189,261.019,399.724,172.293,36.927,156.961
C01207=1052.196,261.267,399.694,172.296,36.930,156.962
C01208=1052.202,261.515,399.665,172.299,36.933,156.962
C01209=1052.208,261.764,399.636,172.302,36.936,156.963
C01210=1052.215,262.012,399.605,172.304,36.939,156.964
C01211=1052.222,262.260,399.576,172.307,36.943,156.965
C01212=1052.228,262.505,399.547,172.310,36.946,156.965
C01213=1052.235,262.750,399.519,172.313,36.949,156.966
C01214=1052.242,262.995,399.490,172.315,36.952,156.967
C01215=1052.248,263.240,399.459,172.318,36.956,156.967
C01216=1052.253,263.484,399.430,172.320,36.959,156.968
C01217=1052.260,263.729,399.401,172.324,36.962,156.969
C01218=1052.266,263.975,399.372,172.326,36.965,156.970
C01219=1052.273,264.219,399.342,172.328,36.969,156.970
C01220=1052.279,264.467,399.313,172.331,36.972,156.971
C01221=1052.285,264.715,399.283,172.333,36.975,156.972
C01222=1052.292,264.964,399.253,172.337,36.979,156.972
C01223=1052.298,265.211,399.224,172.339,36.982,156.973
C01224=1052.304,265.460,399.194,172.342,36.985,156.974
C01225=1052.311,265.708,399.164,172.344,36.989,156.975
C01226=1052.318,265.956,399.134,172.348,36.992,156.975
C01227=1052.324,266.205,399.104,172.350,36.995,156.976
C01228=1052.330,266.452,399.074,172.353,36.999,156.977
C01229=1052.337,266.700,399.045,172.355,37.002,156.978
C01230=1052.343,266.949,399.015,172.359,37.005,156.978
C01231=1052.349,267.196,398.985,172.361,37.008,156.979
C01232=1052.357,267.445,398.955,172.364,37.012,156.980
C01233=1052.362,267.693,398.925,172.366,37.015,156.980
C01234=1052.369,267.941,398.895,172.370,37.018,156.981
C01235=1052.375,268.189,398.865,172.372,37.021,156.982
C01236=1052.381,268.437,398.836,172.375,37.025,156.983
C01237=1052.388,268.686,398.805,172.378,37.028,156.983
C01238=1052.394,268.933,398.775,172.381,37.032,156.984
C01239=1052.401,269.182,398.744,172.383,37.035,156.985
C01240=1052.407,269.429,398.715,172.386,37.038,156.986
C01241=1052.414,269.678,398.685,172.389,37.042,156.986
C01242=1052.420,269.926,398.655,172.392,37.045,156.987
C01243=1052.427,270.174,398.625,172.394,37.048,156.988
C01244=1052.433,270.422,398.594,172.398,37.052,156.989
C01245=1052.439,270.670,398.564,172.400,37.055,156.989
C01246=1052.446,270.918,398.534,172.403,37.058,156.990
C01247=1052.452,271.166,398.503,172.406,37.062,156.991
C01248=1052.459,271.415,398.474,172.409,37.065,156.991
C01249=1052.465,271.663,398.444,172.411,37.068,156.992
C01250=1052.472,271.911,398.414,172.415,37.071,156.993
C01251=1052.478,272.159,398.383,172.417,37.075,156.994
C01252=1052.485,272.407,398.353,172.420,37.078,156.994
C01253=1052.491,272.655,398.323,172.423,37.081,156.995
C01254=1052.497,272.903,398.292,172.426,37.085,156.996
C01255=1052.504,273.151,398.262,172.428,37.088,156.997
C01256=1052.510,273.399,398.232,172.432,37.091,156.997
C01257=1052.516,273.648,398.201,172.434,37.095,156.998
C01258=1052.523,273.894,398.171,172.437,37.098,156.999
C01259=1052.529,274.143,398.140,172.440,37.102,157.000
C01260=1052.535,274.391,398.109,172.443,37.105,157.000
C01261=1052.542,274.639,398.079,172.445,37.108,157.001
C01262=1052.549,274.888,398.049,172.449,37.112,157.002
C01263=1052.555,275.135,398.018,172.451,37.115,157.003
C01264=1052.562,275.384,397.988,172.454,37.119,157.003
C01265=1052.568,275.631,397.958,172.457,37.122,157.004
C01266=1052.574,275.879,397.926,172.460,37.125,157.005
C01267=1052.580,276.127,397.896,172.463,37.128,157.006
C01268=1052.587,276.374,397.866,172.466,37.132,157.006
C01269=1052.594,276.621,397.836,172.468,37.135,157.007
C01270=1052.600,276.869,397.805,172.472,37.138,157.008
C01271=1052.606,277.115,397.775,172.474,37.142,157.009
C01272=1052.613,277.362,397.744,172.477,37.145,157.009
C01273=1052.619,277.609,397.713,172.480,37.149,157.010
C01274=1052.626,277.856,397.683,172.483,37.152,157.011
C01275=1052.633,278.103,397.652,172.486,37.155,157.012
C01276=1052.639,278.350,397.622,172.489,37.159,157.012
C01277=1052.645,278.599,397.591,172.491,37.162,157.013
C01278=1052.652,278.847,397.560,172.495,37.165,157.014
C01279=1052.658,279.095,397.529,172.497,37.169,157.014
C01280=1052.665,279.343,397.499,172.501,37.172,157.015
C01281=1052.671,279.591,397.468,172.503,37.176,157.016
C01282=1052.677,279.839,397.437,172.507,37.179,157.017
C01283=1052.684,280.087,397.406,172.510,37.182,157.018
C01284=1052.690,280.335,397.375,172.512,37.186,157.018
C01285=1052.696,280.582,397.344,172.516,37.189,157.019
C01286=1052.703,280.831,397.313,172.518,37.192,157.020
C01287=1052.710,281.079,397.282,172.522,37.196,157.021
C01288=1052.715,281.327,397.252,172.524,37.199,157.021
C01289=1052.722,281.574,397.220,172.527,37.203,157.022
C01290=1052.729,281.823,397.190,172.530,37.206,157.023
C01291=1052.735,282.070,397.158,172.533,37.210,157.024
C01292=1052.741,282.319,397.128,172.536,37.213,157.025
C01293=1052.748,282.567,397.096,172.539,37.217,157.025
C01294=1052.754,282.814,397.065,172.542,37.220,157.026
C01295=1052.760,283.062,397.035,172.545,37.224,157.027
C01296=1052.767,283.310,397.003,172.548,37.226,157.027
C01297=1052.774,283.558,396.972,172.551,37.230,157.028
C01298=1052.780,283.806,396.941,172.554,37.233,157.029
C01299=1052.786,284.054,396.910,172.557,37.237,157.030
C01300=1052.793,284.302,396.878,172.561,37.240,157.031
C01301=1052.800,284.550,396.848,172.563,37.244,157.031
C01302=1052.806,284.799,396.816,172.567,37.247,157.032
C01303=1052.812,285.046,396.785,172.569,37.251,157.033
C01304=1052.818,285.294,396.753,172.573,37.254,157.034
C01305=1052.825,285.542,396.723,172.575,37.258,157.035
C01306=1052.832,285.790,396.691,172.579,37.261,157.035
C01307=1052.838,286.038,396.660,172.581,37.265,157.036
C01308=1052.845,286.286,396.628,172.585,37.267,157.037
C01309=1052.851,286.533,396.597,172.587,37.271,157.038
C01310=1052.857,286.782,396.566,172.591,37.274,157.038
C01311=1052.864,287.029,396.535,172.594,37.278,157.039
C01312=1052.871,287.277,396.504,172.597,37.281,157.040
C01313=1052.878,287.525,396.472,172.600,37.285,157.041
C01314=1052.884,287.773,396.441,172.603,37.288,157.041
C01315=1052.891,288.021,396.409,172.606,37.292,157.042
C01316=1052.897,288.269,396.378,172.609,37.295,157.043
C01317=1052.903,288.516,396.346,172.612,37.299,157.044
C01318=1052.910,288.764,396.315,172.615,37.302,157.045
C01319=1052.917,289.012,396.283,172.618,37.306,157.045
C01320=1052.923,289.261,396.251,172.622,37.309,157.046
C01321=1052.929,289.508,396.220,172.624,37.312,157.047
C01322=1052.936,289.756,396.188,172.628,37.316,157.048
C01323=1052.943,290.004,396.157,172.631,37.319,157.049
C01324=1052.949,290.262,396.124,172.634,37.323,157.049
C01325=1052.956,290.519,396.091,172.637,37.327,157.050
C01326=1052.962,290.776,396.059,172.641,37.330,157.051
C01327=1052.970,291.032,396.026,172.644,37.334,157.052
C01328=1052.976,291.281,395.994,172.647,37.338,157.053
C01329=1052.982,291.529,395.962,172.650,37.341,157.053
C01330=1052.989,291.776,395.931,172.653,37.345,157.054
C01331=1052.995,292.025,395.899,172.657,37.348,157.055
C01332=1053.002,292.273,395.867,172.659,37.352,157.056
C01333=1053.009,292.520,395.835,172.663,37.355,157.057
C01334=1053.014,292.767,395.803,172.666,37.359,157.057
C01335=1053.021,293.015,395.772,172.669,37.362,157.058
C01336=1053.027,293.263,395.740,172.673,37.365,157.059
C01337=1053.034,293.511,395.708,172.675,37.369,157.060
C01338=1053.041,293.759,395.676,172.679,37.372,157.061
C01339=1053.047,294.007,395.644,172.681,37.376,157.061
C01340=1053.054,294.254,395.612,172.685,37.380,157.062
C01341=1053.060,294.502,395.581,172.689,37.383,157.063
C01342=1053.067,294.751,395.548,172.691,37.387,157.064
C01343=1053.074,294.998,395.516,172.695,37.390,157.065
C01344=1053.080,295.246,395.484,172.697,37.394,157.065
C01345=1053.087,295.494,395.453,172.701,37.397,157.066
C01346=1053.093,295.742,395.420,172.705,37.401,157.067
C01347=1053.100,295.990,395.389,172.707,37.404,157.068
C01348=1053.106,296.237,395.356,172.711,37.408,157.069
C01349=1053.113,296.485,395.324,172.714,37.411,157.070
C01350=1053.119,296.733,395.292,172.717,37.415,157.070
C01351=1053.125,296.981,395.260,172.720,37.419,157.071
C01352=1053.131,297.229,395.227,172.724,37.422,157.072
C01353=1053.138,297.476,395.195,172.727,37.426,157.073
C01354=1053.144,297.724,395.163,172.730,37.430,157.074
C01355=1053.151,297.972,395.130,172.733,37.433,157.075
C01356=1053.157,298.220,395.098,172.737,37.437,157.075
C01357=1053.163,298.468,395.065,172.740,37.441,157.076
C01358=1053.170,298.715,395.033,172.743,37.444,157.077
C01359=1053.176,298.963,395.001,172.746,37.448,157.078
C01360=1053.182,299.211,394.968,172.750,37.451,157.079
C01361=1053.188,299.458,394.936,172.753,37.455,157.080
C01362=1053.194,299.707,394.904,172.756,37.459,157.080
C01363=1053.202,299.954,394.871,172.760,37.462,157.081
C01364=1053.208,300.201,394.839,172.762,37.466,157.082
C01365=1053.215,300.450,394.806,172.766,37.470,157.083
C01366=1053.221,300.697,394.773,172.770,37.473,157.084
C01367=1053.227,300.946,394.741,172.772,37.477,157.085
C01368=1053.234,301.193,394.709,172.776,37.481,157.085
C01369=1053.240,301.440,394.676,172.779,37.484,157.086
C01370=1053.247,301.688,394.643,172.783,37.488,157.087
C01371=1053.253,301.936,394.610,172.786,37.492,157.088
C01372=1053.260,302.184,394.577,172.789,37.496,157.089
C01373=1053.266,302.432,394.545,172.793,37.499,157.090
C01374=1053.273,302.679,394.513,172.796,37.502,157.091
C01375=1053.279,302.927,394.480,172.799,37.506,157.091
C01376=1053.285,303.175,394.448,172.803,37.510,157.092
C01377=1053.292,303.422,394.415,172.806,37.514,157.093
C01378=1053.299,303.670,394.382,172.809,37.517,157.094
C01379=1053.305,303.918,394.349,172.813,37.521,157.095
C01380=1053.312,304.191,394.313,172.816,37.525,157.096
C01381=1053.320,304.464,394.277,172.820,37.529,157.097
C01382=1053.327,304.737,394.241,172.824,37.533,157.098
C01383=1053.334,305.010,394.205,172.827,37.537,157.099
C01384=1053.341,305.258,394.172,172.831,37.541,157.099
C01385=1053.347,305.505,394.139,172.835,37.545,157.100
C01386=1053.353,305.753,394.106,172.838,37.548,157.101
C01387=1053.361,306.001,394.074,172.841,37.552,157.102
C01388=1053.367,306.248,394.040,172.845,37.555,157.103
C01389=1053.374,306.496,394.008,172.848,37.559,157.104
C01390=1053.381,306.744,393.975,172.852,37.563,157.105
C01391=1053.387,306.991,393.942,172.856,37.567,157.106
C01392=1053.393,307.239,393.909,172.858,37.570,157.106
C01393=1053.400,307.487,393.876,172.862,37.574,157.107
C01394=1053.407,307.734,393.843,172.865,37.578,157.108
C01395=1053.414,307.982,393.810,172.869,37.582,157.109
C01396=1053.421,308.230,393.777,172.873,37.585,157.110
C01397=1053.427,308.478,393.745,172.875,37.589,157.111
C01398=1053.434,308.724,393.711,172.879,37.592,157.111
C01399=1053.440,308.973,393.678,172.883,37.596,157.112
C01400=1053.447,309.220,393.645,172.886,37.600,157.113
C01401=1053.454,309.469,393.612,172.890,37.604,157.114
C01402=1053.460,309.716,393.579,172.894,37.607,157.115
C01403=1053.467,309.964,393.546,172.897,37.611,157.116
C01404=1053.473,310.212,393.513,172.900,37.615,157.117
C01405=1053.481,310.459,393.479,172.904,37.619,157.118
C01406=1053.487,310.707,393.446,172.907,37.622,157.118
C01407=1053.495,310.954,393.413,172.911,37.626,157.119
C01408=1053.501,311.202,393.380,172.915,37.629,157.120
C01409=1053.508,311.449,393.346,172.918,37.633,157.121
C01410=1053.515,311.697,393.314,172.922,37.637,157.122
C01411=1053.521,311.945,393.281,172.925,37.641,157.123
C01412=1053.528,312.192,393.247,172.928,37.645,157.124
C01413=1053.535,312.441,393.214,172.932,37.648,157.125
C01414=1053.542,312.688,393.181,172.936,37.652,157.125
C01415=1053.548,312.936,393.148,172.939,37.656,157.126
C01416=1053.555,313.183,393.114,172.943,37.659,157.127
C01417=1053.562,313.430,393.080,172.947,37.663,157.128
C01418=1053.568,313.678,393.047,172.950,37.667,157.129
C01419=1053.575,313.926,393.013,172.954,37.671,157.130
C01420=1053.581,314.173,392.979,172.957,37.675,157.131
C01421=1053.588,314.422,392.946,172.960,37.679,157.132
C01422=1053.594,314.669,392.912,172.964,37.683,157.133
C01423=1053.601,314.917,392.878,172.968,37.687,157.134
C01424=1053.607,315.164,392.844,172.971,37.690,157.135
C01425=1053.614,315.412,392.810,172.975,37.694,157.136
C01426=1053.619,315.659,392.777,172.979,37.698,157.136
C01427=1053.627,315.907,392.743,172.983,37.702,157.137
C01428=1053.633,316.154,392.709,172.986,37.706,157.138
C01429=1053.640,316.402,392.675,172.989,37.710,157.139
C01430=1053.646,316.649,392.641,172.993,37.714,157.140
C01431=1053.653,316.897,392.607,172.996,37.718,157.141
C01432=1053.659,317.145,392.573,173.000,37.722,157.142
C01433=1053.666,317.392,392.539,173.004,37.726,157.143
C01434=1053.672,317.641,392.506,173.008,37.730,157.144
C01435=1053.679,317.888,392.472,173.011,37.734,157.145
C01436=1053.686,318.165,392.434,173.015,37.738,157.146
C01437=1053.693,318.443,392.396,173.020,37.742,157.147
C01438=1053.702,318.720,392.357,173.024,37.747,157.148
C01439=1053.708,318.996,392.319,173.028,37.752,157.149
C01440=1053.715,319.244,392.285,173.031,37.755,157.150
C01441=1053.722,319.492,392.251,173.035,37.759,157.151
C01442=1053.728,319.739,392.217,173.039,37.763,157.152
C01443=1053.735,319.987,392.183,173.042,37.767,157.153
C01444=1053.742,320.235,392.149,173.046,37.771,157.154
C01445=1053.747,320.482,392.115,173.050,37.775,157.155
C01446=1053.755,320.730,392.081,173.054,37.779,157.156
C01447=1053.761,320.978,392.046,173.057,37.783,157.157
C01448=1053.769,321.225,392.012,173.061,37.787,157.158
C01449=1053.774,321.472,391.978,173.065,37.791,157.158
C01450=1053.782,321.720,391.944,173.068,37.795,157.159
C01451=1053.788,321.968,391.910,173.072,37.799,157.160
C01452=1053.795,322.215,391.876,173.076,37.803,157.161
C01453=1053.802,322.463,391.841,173.080,37.807,157.162
C01454=1053.808,322.710,391.807,173.084,37.811,157.163
C01455=1053.815,322.958,391.773,173.087,37.815,157.164
C01456=1053.822,323.206,391.738,173.091,37.819,157.165
C01457=1053.829,323.453,391.704,173.095,37.823,157.166
C01458=1053.836,323.701,391.669,173.098,37.827,157.167
C01459=1053.841,323.948,391.635,173.102,37.831,157.168
C01460=1053.849,324.195,391.601,173.106,37.835,157.169
C01461=1053.855,324.443,391.566,173.110,37.839,157.170
C01462=1053.863,324.690,391.532,173.113,37.843,157.171
C01463=1053.869,324.938,391.497,173.117,37.847,157.172
C01464=1053.876,325.186,391.463,173.122,37.851,157.173
C01465=1053.883,325.433,391.428,173.126,37.855,157.174
C01466=1053.890,325.681,391.394,173.130,37.860,157.175
C01467=1053.897,325.928,391.359,173.133,37.864,157.176
C01468=1053.904,326.176,391.325,173.137,37.867,157.177
C01469=1053.911,326.424,391.290,173.141,37.871,157.178
C01470=1053.918,326.671,391.256,173.145,37.875,157.179
C01471=1053.925,326.919,391.221,173.148,37.880,157.180
C01472=1053.931,327.166,391.186,173.152,37.884,157.181
C01473=1053.939,327.414,391.152,173.156,37.888,157.182
C01474=1053.945,327.661,391.117,173.160,37.892,157.183
C01475=1053.952,327.909,391.082,173.164,37.896,157.184
C01476=1053.959,328.156,391.048,173.168,37.900,157.185
C01477=1053.966,328.403,391.013,173.172,37.904,157.186
C01478=1053.972,328.651,390.978,173.176,37.908,157.187
C01479=1053.980,328.898,390.944,173.180,37.912,157.188
C01480=1053.987,329.146,390.909,173.183,37.916,157.189
C01481=1053.993,329.394,390.874,173.187,37.921,157.190
C01482=1054.001,329.641,390.840,173.192,37.925,157.191
C01483=1054.007,329.888,390.805,173.196,37.929,157.192
C01484=1054.014,330.136,390.769,173.199,37.933,157.193
C01485=1054.021,330.383,390.734,173.203,37.937,157.194
C01486=1054.028,330.630,390.699,173.207,37.941,157.195
C01487=1054.034,330.878,390.665,173.211,37.945,157.196
C01488=1054.041,331.126,390.630,173.216,37.950,157.197
C01489=1054.048,331.373,390.594,173.219,37.954,157.198
C01490=1054.055,331.620,390.559,173.223,37.958,157.199
C01491=1054.061,331.868,390.524,173.227,37.963,157.200
C01492=1054.067,332.091,390.492,173.231,37.966,157.201
C01493=1054.074,332.313,390.461,173.235,37.970,157.202
C01494=1054.080,332.536,390.428,173.238,37.974,157.203
C01495=1054.086,332.759,390.397,173.241,37.978,157.204
C01496=1054.093,332.982,390.365,173.245,37.982,157.205
C01497=1054.098,333.204,390.334,173.249,37.986,157.205
C01498=1054.104,333.427,390.302,173.252,37.989,157.206
C01499=1054.111,333.649,390.270,173.256,37.993,157.207
C01500=1054.117,333.897,390.234,173.260,37.997,157.208
C01501=1054.124,334.144,390.199,173.264,38.002,157.209
C01502=1054.131,334.393,390.164,173.269,38.006,157.211
C01503=1054.138,334.639,390.128,173.272,38.010,157.211
C01504=1054.145,334.887,390.093,173.276,38.015,157.213
C01505=1054.152,335.134,390.058,173.280,38.019,157.214
C01506=1054.158,335.381,390.023,173.284,38.023,157.215
C01507=1054.166,335.629,389.987,173.289,38.027,157.216
C01508=1054.173,335.876,389.951,173.293,38.032,157.217
C01509=1054.180,336.124,389.916,173.297,38.036,157.218
C01510=1054.186,336.371,389.880,173.300,38.041,157.219
C01511=1054.193,336.619,389.844,173.305,38.045,157.220
C01512=1054.200,336.866,389.809,173.309,38.049,157.221
C01513=1054.207,337.113,389.774,173.313,38.054,157.222
C01514=1054.213,337.360,389.737,173.317,38.058,157.223
C01515=1054.221,337.609,389.702,173.322,38.062,157.224
C01516=1054.228,337.855,389.666,173.326,38.067,157.225
C01517=1054.234,338.103,389.630,173.329,38.071,157.226
C01518=1054.241,338.350,389.594,173.334,38.076,157.228
C01519=1054.248,338.598,389.559,173.338,38.080,157.229
C01520=1054.255,338.845,389.522,173.342,38.085,157.230
C01521=1054.261,339.092,389.487,173.346,38.089,157.231
C01522=1054.269,339.340,389.451,173.351,38.094,157.232
C01523=1054.275,339.587,389.415,173.355,38.098,157.233
C01524=1054.282,339.834,389.380,173.359,38.102,157.234
C01525=1054.290,340.081,389.343,173.364,38.107,157.235
C01526=1054.296,340.329,389.308,173.367,38.111,157.236
C01527=1054.303,340.576,389.272,173.371,38.116,157.237
C01528=1054.311,340.823,389.236,173.376,38.120,157.239
C01529=1054.317,341.071,389.200,173.380,38.125,157.240
C01530=1054.324,341.318,389.164,173.384,38.130,157.241
C01531=1054.331,341.566,389.127,173.389,38.134,157.242
C01532=1054.338,341.812,389.091,173.393,38.139,157.243
C01533=1054.345,342.060,389.055,173.397,38.143,157.244
C01534=1054.351,342.307,389.019,173.402,38.147,157.245
C01535=1054.359,342.555,388.983,173.406,38.152,157.246
C01536=1054.366,342.802,388.947,173.410,38.156,157.247
C01537=1054.373,343.049,388.910,173.415,38.161,157.249
C01538=1054.379,343.296,388.874,173.418,38.166,157.250
C01539=1054.387,343.544,388.838,173.423,38.170,157.251
C01540=1054.393,343.791,388.801,173.427,38.175,157.252
C01541=1054.400,344.038,388.766,173.431,38.180,157.253
C01542=1054.407,344.285,388.729,173.436,38.184,157.254
C01543=1054.414,344.532,388.693,173.440,38.189,157.256
C01544=1054.421,344.780,388.656,173.445,38.193,157.257
C01545=1054.428,345.027,388.620,173.449,38.198,157.258
C01546=1054.435,345.274,388.583,173.453,38.203,157.259
C01547=1054.446,345.670,388.525,173.461,38.210,157.261
C01548=1054.458,346.086,388.463,173.468,38.218,157.263
C01549=1054.465,346.353,388.424,173.472,38.223,157.264
C01550=1054.473,346.621,388.384,173.477,38.228,157.265
C01551=1054.481,346.889,388.344,173.482,38.233,157.267
C01552=1054.488,347.136,388.308,173.486,38.238,157.268
C01553=1054.494,347.384,388.271,173.491,38.243,157.269
C01554=1054.502,347.631,388.235,173.495,38.248,157.270
C01555=1054.509,347.877,388.198,173.499,38.252,157.271
C01556=1054.516,348.125,388.161,173.504,38.257,157.273
C01557=1054.523,348.373,388.124,173.508,38.261,157.274
C01558=1054.530,348.619,388.088,173.513,38.266,157.275
C01559=1054.537,348.867,388.051,173.517,38.271,157.276
C01560=1054.544,349.115,388.014,173.522,38.276,157.277
C01561=1054.551,349.361,387.977,173.526,38.281,157.279
C01562=1054.558,349.608,387.941,173.531,38.286,157.280
C01563=1054.565,349.856,387.903,173.535,38.290,157.281
C01564=1054.572,350.103,387.867,173.540,38.295,157.282
C01565=1054.579,350.350,387.829,173.544,38.300,157.283
C01566=1054.587,350.597,387.793,173.549,38.304,157.284
C01567=1054.594,350.844,387.755,173.553,38.309,157.286
C01568=1054.600,351.091,387.719,173.558,38.314,157.287
C01569=1054.608,351.339,387.681,173.562,38.319,157.288
C01570=1054.615,351.586,387.644,173.567,38.324,157.289
C01571=1054.621,351.833,387.607,173.572,38.328,157.291
C01572=1054.628,352.080,387.570,173.576,38.333,157.292
C01573=1054.636,352.327,387.532,173.581,38.338,157.293
C01574=1054.643,352.574,387.496,173.585,38.343,157.294
C01575=1054.650,352.821,387.459,173.590,38.348,157.296
C01576=1054.657,353.068,387.422,173.594,38.353,157.297
C01577=1054.664,353.315,387.384,173.600,38.358,157.298
C01578=1054.672,353.562,387.346,173.604,38.363,157.299
C01579=1054.679,353.810,387.310,173.609,38.368,157.301
C01580=1054.685,354.056,387.272,173.614,38.373,157.302
C01581=1054.692,354.304,387.235,173.618,38.378,157.303
C01582=1054.700,354.551,387.197,173.623,38.383,157.304
C01583=1054.707,354.798,387.160,173.627,38.388,157.306
C01584=1054.714,355.045,387.122,173.632,38.393,157.307
C01585=1054.721,355.292,387.085,173.637,38.398,157.308
C01586=1054.729,355.539,387.047,173.641,38.403,157.309
C01587=1054.736,355.786,387.010,173.646,38.408,157.311
C01588=1054.742,356.033,386.972,173.650,38.413,157.312
C01589=1054.749,356.280,386.935,173.655,38.418,157.313
C01590=1054.756,356.527,386.897,173.660,38.423,157.315
C01591=1054.764,356.775,386.859,173.665,38.428,157.316
C01592=1054.771,357.022,386.822,173.670,38.433,157.317
C01593=1054.778,357.269,386.784,173.675,38.438,157.318
C01594=1054.786,357.515,386.746,173.679,38.443,157.320
C01595=1054.793,357.762,386.709,173.684,38.449,157.321
C01596=1054.800,358.010,386.671,173.689,38.454,157.322
C01597=1054.807,358.257,386.634,173.693,38.459,157.324
C01598=1054.815,358.503,386.595,173.698,38.464,157.325
C01599=1054.821,358.751,386.557,173.703,38.469,157.326
C01600=1054.829,358.998,386.520,173.708,38.474,157.328
C01601=1054.836,359.244,386.481,173.713,38.479,157.329
C01602=1054.843,359.491,386.444,173.718,38.485,157.330
C01603=1054.850,359.739,386.406,173.722,38.490,157.332
C01604=1054.859,360.012,386.363,173.727,38.496,157.333
C01605=1054.867,360.284,386.322,173.734,38.501,157.334
C01606=1054.874,360.557,386.280,173.739,38.507,157.336
C01607=1054.883,360.830,386.238,173.744,38.513,157.337
C01608=1054.890,361.077,386.199,173.749,38.518,157.339
C01609=1054.897,361.324,386.162,173.753,38.524,157.340
C01610=1054.904,361.571,386.124,173.759,38.528,157.341
C01611=1054.911,361.818,386.085,173.764,38.534,157.343
C01612=1054.918,362.065,386.047,173.769,38.539,157.344
C01613=1054.927,362.312,386.009,173.773,38.544,157.346
C01614=1054.934,362.559,385.971,173.778,38.550,157.347
C01615=1054.941,362.806,385.932,173.784,38.555,157.348
C01616=1054.948,363.053,385.894,173.789,38.560,157.350
C01617=1054.956,363.299,385.856,173.793,38.565,157.351
C01618=1054.963,363.547,385.817,173.798,38.571,157.352
C01619=1054.970,363.794,385.779,173.803,38.576,157.354
C01620=1054.977,364.041,385.740,173.808,38.582,157.355
C01621=1054.985,364.287,385.702,173.813,38.587,157.357
C01622=1054.992,364.534,385.663,173.818,38.593,157.358
C01623=1054.998,364.781,385.624,173.823,38.598,157.359
C01624=1055.007,365.028,385.586,173.828,38.604,157.361
C01625=1055.013,365.275,385.548,173.834,38.609,157.362
C01626=1055.021,365.522,385.509,173.839,38.614,157.364
C01627=1055.027,365.769,385.471,173.843,38.620,157.365
C01628=1055.036,366.016,385.432,173.848,38.625,157.367
C01629=1055.043,366.262,385.392,173.854,38.631,157.368
C01630=1055.049,366.509,385.354,173.859,38.636,157.369
C01631=1055.057,366.756,385.315,173.864,38.642,157.371
C01632=1055.064,367.003,385.276,173.869,38.648,157.372
C01633=1055.072,367.250,385.238,173.874,38.653,157.374
C01634=1055.079,367.496,385.199,173.879,38.658,157.375
C01635=1055.087,367.744,385.160,173.884,38.664,157.377
C01636=1055.094,367.990,385.122,173.889,38.670,157.378
C01637=1055.102,368.237,385.082,173.895,38.675,157.379
C01638=1055.109,368.484,385.043,173.900,38.681,157.381
C01639=1055.116,368.731,385.005,173.905,38.686,157.382
C01640=1055.124,368.978,384.965,173.911,38.692,157.384
C01641=1055.131,369.224,384.926,173.916,38.697,157.385
C01642=1055.139,369.472,384.887,173.921,38.703,157.387
C01643=1055.146,369.717,384.848,173.925,38.709,157.388
C01644=1055.153,369.964,384.809,173.931,38.714,157.390
C01645=1055.161,370.212,384.770,173.936,38.720,157.391
C01646=1055.168,370.458,384.731,173.941,38.726,157.393
C01647=1055.176,370.705,384.692,173.947,38.732,157.394
C01648=1055.183,370.951,384.653,173.952,38.737,157.396
C01649=1055.191,371.199,384.614,173.957,38.743,157.397
C01650=1055.198,371.445,384.574,173.963,38.748,157.399
C01651=1055.206,371.692,384.536,173.968,38.754,157.400
C01652=1055.214,371.939,384.496,173.973,38.760,157.402
C01653=1055.221,372.185,384.456,173.979,38.766,157.403
C01654=1055.229,372.433,384.417,173.984,38.772,157.405
C01655=1055.236,372.679,384.378,173.989,38.778,157.406
C01656=1055.244,372.926,384.338,173.995,38.783,157.408
C01657=1055.251,373.172,384.298,174.000,38.789,157.409
C01658=1055.258,373.420,384.259,174.005,38.795,157.411
C01659=1055.265,373.666,384.219,174.011,38.801,157.412
C01660=1055.274,373.957,384.173,174.018,38.808,157.414
C01661=1055.283,374.249,384.125,174.024,38.815,157.416
C01662=1055.292,374.540,384.079,174.030,38.822,157.418
C01663=1055.301,374.832,384.032,174.036,38.829,157.420
C01664=1055.309,375.079,383.992,174.042,38.835,157.421
C01665=1055.316,375.326,383.953,174.047,38.841,157.423
C01666=1055.323,375.572,383.913,174.053,38.847,157.424
C01667=1055.331,375.819,383.873,174.058,38.852,157.426
C01668=1055.339,376.066,383.833,174.064,38.858,157.428
C01669=1055.346,376.311,383.793,174.070,38.865,157.429
C01670=1055.354,376.558,383.753,174.075,38.871,157.431
C01671=1055.362,376.805,383.713,174.081,38.877,157.432
C01672=1055.369,377.051,383.673,174.086,38.883,157.434
C01673=1055.377,377.298,383.634,174.092,38.889,157.436
C01674=1055.384,377.545,383.594,174.097,38.895,157.437
C01675=1055.392,377.791,383.553,174.103,38.901,157.439
C01676=1055.400,378.038,383.513,174.108,38.907,157.440
C01677=1055.407,378.285,383.474,174.115,38.913,157.442
C01678=1055.415,378.531,383.434,174.120,38.919,157.444
C01679=1055.423,378.778,383.393,174.126,38.925,157.445
C01680=1055.431,379.025,383.353,174.131,38.931,157.447
C01681=1055.438,379.272,383.313,174.137,38.937,157.449
C01682=1055.446,379.518,383.272,174.142,38.944,157.450
C01683=1055.454,379.765,383.233,174.149,38.950,157.452
C01684=1055.462,380.011,383.192,174.154,38.956,157.454
C01685=1055.469,380.257,383.152,174.160,38.962,157.455
C01686=1055.477,380.504,383.111,174.165,38.968,157.457
C01687=1055.484,380.751,383.071,174.171,38.975,157.459
C01688=1055.492,380.997,383.031,174.177,38.981,157.460
C01689=1055.500,381.244,382.989,174.183,38.987,157.462
C01690=1055.507,381.491,382.949,174.188,38.994,157.464
C01691=1055.515,381.737,382.909,174.194,39.000,157.465
C01692=1055.523,381.983,382.868,174.199,39.007,157.467
C01693=1055.531,382.230,382.827,174.206,39.013,157.469
C01694=1055.538,382.477,382.786,174.212,39.019,157.470
C01695=1055.546,382.723,382.746,174.217,39.025,157.472
C01696=1055.554,382.969,382.705,174.223,39.032,157.474
C01697=1055.561,383.216,382.664,174.229,39.038,157.476
C01698=1055.569,383.462,382.623,174.235,39.044,157.477
C01699=1055.577,383.709,382.583,174.241,39.051,157.479
C01700=1055.584,383.955,382.541,174.247,39.058,157.481
C01701=1055.592,384.202,382.501,174.253,39.064,157.483
C01702=1055.600,384.448,382.460,174.258,39.071,157.484
C01703=1055.608,384.694,382.419,174.264,39.077,157.486
C01704=1055.616,384.941,382.378,174.271,39.083,157.488
C01705=1055.623,385.187,382.337,174.276,39.090,157.490
C01706=1055.631,385.434,382.296,174.282,39.097,157.491
C01707=1055.639,385.680,382.256,174.289,39.103,157.493
C01708=1055.646,385.926,382.215,174.294,39.110,157.495
C01709=1055.655,386.173,382.174,174.301,39.117,157.497
C01710=1055.663,386.419,382.132,174.307,39.123,157.499
C01711=1055.671,386.666,382.091,174.312,39.129,157.500
C01712=1055.679,386.912,382.050,174.319,39.136,157.502
C01713=1055.686,387.159,382.009,174.325,39.143,157.504
C01714=1055.695,387.405,381.967,174.331,39.150,157.506
C01715=1055.702,387.652,381.926,174.337,39.156,157.508
C01716=1055.713,387.975,381.873,174.345,39.165,157.510
C01717=1055.723,388.298,381.818,174.353,39.173,157.512
C01718=1055.734,388.621,381.764,174.361,39.183,157.515
C01719=1055.744,388.944,381.709,174.369,39.192,157.517
C01720=1055.752,389.191,381.669,174.376,39.198,157.519
C01721=1055.761,389.437,381.626,174.381,39.205,157.521
C01722=1055.769,389.684,381.586,174.388,39.212,157.523
C01723=1055.777,389.930,381.543,174.394,39.219,157.525
C01724=1055.784,390.176,381.501,174.401,39.225,157.527
C01725=1055.792,390.422,381.461,174.407,39.232,157.528
C01726=1055.801,390.669,381.418,174.413,39.239,157.530
C01727=1055.808,390.915,381.377,174.419,39.246,157.532
C01728=1055.816,391.161,381.335,174.426,39.253,157.534
C01729=1055.825,391.407,381.293,174.432,39.260,157.536
C01730=1055.832,391.654,381.252,174.438,39.267,157.538
C01731=1055.840,391.901,381.209,174.444,39.274,157.540
C01732=1055.849,392.146,381.168,174.451,39.281,157.542
C01733=1055.857,392.393,381.126,174.457,39.288,157.544
C01734=1055.864,392.639,381.084,174.464,39.295,157.546
C01735=1055.873,392.886,381.041,174.471,39.302,157.547
C01736=1055.881,393.131,381.000,174.477,39.309,157.550
C01737=1055.889,393.378,380.958,174.483,39.316,157.551
C01738=1055.897,393.624,380.916,174.489,39.324,157.553
C01739=1055.905,393.870,380.873,174.496,39.330,157.555
C01740=1055.913,394.116,380.831,174.503,39.338,157.557
C01741=1055.921,394.363,380.789,174.509,39.345,157.559
C01742=1055.929,394.609,380.747,174.516,39.352,157.561
C01743=1055.937,394.855,380.704,174.522,39.359,157.563
C01744=1055.946,395.101,380.662,174.529,39.366,157.565
C01745=1055.954,395.347,380.620,174.536,39.374,157.567
C01746=1055.962,395.594,380.578,174.541,39.381,157.569
C01747=1055.970,395.840,380.535,174.548,39.388,157.571
C01748=1055.978,396.086,380.493,174.555,39.395,157.573
C01749=1055.986,396.332,380.450,174.561,39.403,157.575
C01750=1055.995,396.579,380.407,174.568,39.410,157.577
C01751=1056.002,396.824,380.365,174.575,39.417,157.579
C01752=1056.011,397.071,380.322,174.582,39.425,157.582
C01753=1056.019,397.317,380.279,174.588,39.432,157.584
C01754=1056.027,397.563,380.237,174.595,39.440,157.586
C01755=1056.035,397.809,380.194,174.602,39.447,157.588
C01756=1056.044,398.055,380.151,174.608,39.454,157.590
C01757=1056.052,398.301,380.109,174.615,39.462,157.592
C01758=1056.060,398.547,380.066,174.622,39.470,157.594
C01759=1056.068,398.794,380.022,174.629,39.477,157.596
C01760=1056.076,399.039,379.980,174.635,39.484,157.598
C01761=1056.084,399.286,379.937,174.642,39.492,157.600
C01762=1056.093,399.532,379.894,174.649,39.500,157.602
C01763=1056.101,399.778,379.851,174.656,39.507,157.604
C01764=1056.110,400.024,379.808,174.664,39.515,157.607
C01765=1056.118,400.270,379.765,174.670,39.522,157.609
C01766=1056.127,400.516,379.722,174.677,39.530,157.611
C01767=1056.135,400.762,379.679,174.684,39.537,157.613
C01768=1056.143,401.008,379.636,174.691,39.545,157.615
C01769=1056.152,401.255,379.593,174.698,39.553,157.617
C01770=1056.160,401.501,379.549,174.705,39.560,157.620
C01771=1056.169,401.747,379.506,174.712,39.568,157.622
C01772=1056.180,402.088,379.446,174.721,39.579,157.625
C01773=1056.192,402.429,379.386,174.731,39.590,157.628
C01774=1056.203,402.770,379.326,174.741,39.601,157.631
C01775=1056.215,403.111,379.265,174.751,39.612,157.634
C01776=1056.223,403.357,379.222,174.759,39.619,157.636
C01777=1056.232,403.604,379.178,174.766,39.627,157.638
C01778=1056.241,403.849,379.134,174.773,39.635,157.641
C01779=1056.249,404.095,379.091,174.780,39.644,157.643
C01780=1056.257,404.341,379.047,174.787,39.651,157.645
C01781=1056.266,404.587,379.004,174.795,39.659,157.648
C01782=1056.274,404.833,378.959,174.802,39.668,157.650
C01783=1056.283,405.079,378.916,174.809,39.675,157.652
C01784=1056.291,405.325,378.872,174.816,39.683,157.654
C01785=1056.300,405.571,378.828,174.824,39.692,157.657
C01786=1056.308,405.817,378.784,174.831,39.700,157.659
C01787=1056.317,406.063,378.740,174.838,39.708,157.661
C01788=1056.325,406.309,378.696,174.846,39.716,157.664
C01789=1056.333,406.555,378.652,174.853,39.724,157.666
C01790=1056.342,406.801,378.608,174.860,39.732,157.668
C01791=1056.350,407.047,378.563,174.868,39.741,157.671
C01792=1056.359,407.292,378.520,174.875,39.749,157.673
C01793=1056.368,407.538,378.475,174.882,39.757,157.675
C01794=1056.376,407.784,378.431,174.890,39.766,157.678
C01795=1056.385,408.030,378.386,174.898,39.774,157.680
C01796=1056.393,408.276,378.342,174.906,39.782,157.683
C01797=1056.402,408.521,378.298,174.913,39.790,157.685
C01798=1056.411,408.768,378.254,174.920,39.799,157.687
C01799=1056.419,409.014,378.209,174.928,39.807,157.690
C01800=1056.428,409.260,378.165,174.935,39.815,157.692
C01801=1056.437,409.506,378.121,174.944,39.824,157.695
C01802=1056.445,409.751,378.075,174.951,39.832,157.697
C01803=1056.455,409.998,378.031,174.959,39.841,157.700
C01804=1056.463,410.243,377.987,174.966,39.850,157.702
C01805=1056.472,410.489,377.942,174.975,39.858,157.704
C01806=1056.481,410.735,377.898,174.982,39.867,157.707
C01807=1056.490,410.980,377.852,174.990,39.875,157.709
C01808=1056.498,411.227,377.808,174.998,39.884,157.712
C01809=1056.506,411.473,377.763,175.006,39.892,157.714
C01810=1056.516,411.718,377.719,175.013,39.901,157.717
C01811=1056.525,411.964,377.673,175.022,39.910,157.719
C01812=1056.534,412.210,377.628,175.029,39.918,157.722
C01813=1056.543,412.455,377.584,175.037,39.927,157.724
C01814=1056.552,412.702,377.539,175.045,39.935,157.727
C01815=1056.561,412.947,377.494,175.053,39.944,157.730
C01816=1056.570,413.193,377.448,175.062,39.953,157.732
C01817=1056.579,413.439,377.404,175.069,39.962,157.735
C01818=1056.588,413.685,377.359,175.077,39.970,157.737
